DATA_BLOCK "COM_SHUTTLE"	// DB 200
VERSION : 0.1
  STRUCT
   DB_VAR : INT  := 300;	//Temporary placeholder variable
   DB_VAR1 : INT  := 300;	//Temporary placeholder variable
   DB_VAR2 : INT  := 300;	//Temporary placeholder variable
   DB_VAR3 : INT  := 300;	//Temporary placeholder variable
   DB_VAR4 : INT  := 300;	//Temporary placeholder variable
   DB_VAR5 : INT  := 300;	//Temporary placeholder variable
   DB_VAR6 : INT  := 300;	//Temporary placeholder variable
   DB_VAR7 : INT  := 300;	//Temporary placeholder variable
   DB_VAR8 : INT  := 300;	//Temporary placeholder variable
   DB_VAR9 : INT  := 300;	//Temporary placeholder variable
   DB_VAR10 : INT  := 300;	//Temporary placeholder variable
   DB_VAR11 : INT  := 300;	//Temporary placeholder variable
   DB_VAR12 : INT  := 300;	//Temporary placeholder variable
   DB_VAR13 : INT  := 300;	//Temporary placeholder variable
   DB_VAR14 : INT  := 300;	//Temporary placeholder variable
   DB_VAR15 : INT  := 300;	//Temporary placeholder variable
   DB_VAR16 : INT  := 300;	//Temporary placeholder variable
   DB_VAR17 : INT  := 300;	//Temporary placeholder variable
   DB_VAR18 : INT  := 300;	//Temporary placeholder variable
   DB_VAR19 : INT  := 300;	//Temporary placeholder variable
   DB_VAR20 : INT  := 300;	//Temporary placeholder variable
   DB_VAR21 : INT  := 300;	//Temporary placeholder variable
   DB_VAR22 : INT  := 300;	//Temporary placeholder variable
   DB_VAR23 : INT  := 300;	//Temporary placeholder variable
   DB_VAR24 : INT  := 300;	//Temporary placeholder variable
   DB_VAR25 : INT  := 300;	//Temporary placeholder variable
   DB_VAR26 : INT  := 300;	//Temporary placeholder variable
   DB_VAR27 : INT  := 300;	//Temporary placeholder variable
   DB_VAR28 : INT  := 300;	//Temporary placeholder variable
   DB_VAR29 : INT  := 300;	//Temporary placeholder variable
   DB_VAR30 : INT  := 300;	//Temporary placeholder variable
   DB_VAR31 : INT  := 300;	//Temporary placeholder variable
   DB_VAR32 : INT  := 300;	//Temporary placeholder variable
   DB_VAR33 : INT  := 300;	//Temporary placeholder variable
   DB_VAR34 : INT  := 300;	//Temporary placeholder variable
   DB_VAR35 : INT  := 300;	//Temporary placeholder variable
   DB_VAR36 : INT  := 300;	//Temporary placeholder variable
   DB_VAR37 : INT  := 300;	//Temporary placeholder variable
   DB_VAR38 : INT  := 300;	//Temporary placeholder variable
   DB_VAR39 : INT  := 300;	//Temporary placeholder variable
   DB_VAR40 : INT  := 300;	//Temporary placeholder variable
   DB_VAR41 : INT  := 300;	//Temporary placeholder variable
   DB_VAR42 : INT  := 300;	//Temporary placeholder variable
   DB_VAR43 : INT  := 300;	//Temporary placeholder variable
   DB_VAR44 : INT  := 300;	//Temporary placeholder variable
   DB_VAR45 : INT  := 300;	//Temporary placeholder variable
   DB_VAR46 : INT  := 300;	//Temporary placeholder variable
   DB_VAR47 : INT  := 300;	//Temporary placeholder variable
   DB_VAR48 : INT  := 300;	//Temporary placeholder variable
   DB_VAR49 : INT  := 300;	//Temporary placeholder variable
   DB_VAR50 : INT  := 300;	//Temporary placeholder variable
   DB_VAR51 : INT  := 300;	//Temporary placeholder variable
   DB_VAR52 : INT  := 300;	//Temporary placeholder variable
   DB_VAR53 : INT  := 300;	//Temporary placeholder variable
   DB_VAR54 : INT  := 300;	//Temporary placeholder variable
   DB_VAR55 : INT  := 300;	//Temporary placeholder variable
   DB_VAR56 : INT  := 300;	//Temporary placeholder variable
   DB_VAR57 : INT  := 300;	//Temporary placeholder variable
   DB_VAR58 : INT  := 300;	//Temporary placeholder variable
   DB_VAR59 : INT  := 300;	//Temporary placeholder variable
   DB_VAR60 : INT  := 300;	//Temporary placeholder variable
   DB_VAR61 : INT  := 300;	//Temporary placeholder variable
   DB_VAR62 : INT  := 300;	//Temporary placeholder variable
   DB_VAR63 : INT  := 300;	//Temporary placeholder variable
   DB_VAR64 : INT  := 300;	//Temporary placeholder variable
   DB_VAR65 : INT  := 300;	//Temporary placeholder variable
   DB_VAR66 : INT  := 300;	//Temporary placeholder variable
   DB_VAR67 : INT  := 300;	//Temporary placeholder variable
   DB_VAR68 : INT  := 300;	//Temporary placeholder variable
   DB_VAR69 : INT  := 300;	//Temporary placeholder variable
   DB_VAR70 : INT  := 300;	//Temporary placeholder variable
   DB_VAR71 : INT  := 300;	//Temporary placeholder variable
   DB_VAR72 : INT  := 300;	//Temporary placeholder variable
   DB_VAR73 : INT  := 300;	//Temporary placeholder variable
   DB_VAR74 : INT  := 300;	//Temporary placeholder variable
   DB_VAR75 : INT  := 300;	//Temporary placeholder variable
   DB_VAR76 : INT  := 300;	//Temporary placeholder variable
   DB_VAR77 : INT  := 300;	//Temporary placeholder variable
   DB_VAR78 : INT  := 300;	//Temporary placeholder variable
   DB_VAR79 : INT  := 300;	//Temporary placeholder variable
   DB_VAR80 : INT  := 300;	//Temporary placeholder variable
   DB_VAR81 : INT  := 300;	//Temporary placeholder variable
   DB_VAR82 : INT  := 300;	//Temporary placeholder variable
   DB_VAR83 : INT  := 300;	//Temporary placeholder variable
   DB_VAR84 : INT  := 300;	//Temporary placeholder variable
   DB_VAR85 : INT  := 300;	//Temporary placeholder variable
   DB_VAR86 : INT  := 300;	//Temporary placeholder variable
   DB_VAR87 : INT  := 300;	//Temporary placeholder variable
   DB_VAR88 : INT  := 300;	//Temporary placeholder variable
   DB_VAR89 : INT  := 300;	//Temporary placeholder variable
   DB_VAR90 : INT  := 300;	//Temporary placeholder variable
   DB_VAR91 : INT  := 300;	//Temporary placeholder variable
   DB_VAR92 : INT  := 300;	//Temporary placeholder variable
   DB_VAR93 : INT  := 300;	//Temporary placeholder variable
   DB_VAR94 : INT  := 300;	//Temporary placeholder variable
   DB_VAR95 : INT  := 300;	//Temporary placeholder variable
   DB_VAR96 : INT  := 300;	//Temporary placeholder variable
   DB_VAR97 : INT  := 300;	//Temporary placeholder variable
   DB_VAR98 : INT  := 300;	//Temporary placeholder variable
   DB_VAR99 : INT  := 300;	//Temporary placeholder variable
  END_STRUCT ;	
BEGIN
   DB_VAR := 324;
   DB_VAR1 := 3242;
   DB_VAR2 := 2;
   DB_VAR3 := 2;
   DB_VAR4 := 55;
   DB_VAR5 := 1;
   DB_VAR6 := 1;
   DB_VAR7 := 1;
   DB_VAR8 := 1;
   DB_VAR9 := 23423;
   DB_VAR10 := 1;
   DB_VAR11 := 1;
   DB_VAR12 := 1;
   DB_VAR13 := 1;
   DB_VAR14 := 1;
   DB_VAR15 := 2;
   DB_VAR16 := 333;
   DB_VAR17 := 3;
   DB_VAR18 := 300;
   DB_VAR19 := 33;
   DB_VAR20 := 300;
   DB_VAR21 := 8;
   DB_VAR22 := 300;
   DB_VAR23 := 300;
   DB_VAR24 := 300;
   DB_VAR25 := 300;
   DB_VAR26 := 300;
   DB_VAR27 := 4;
   DB_VAR28 := 333;
   DB_VAR29 := 300;
   DB_VAR30 := 300;
   DB_VAR31 := 3;
   DB_VAR32 := 300;
   DB_VAR33 := 300;
   DB_VAR34 := 300;
   DB_VAR35 := 300;
   DB_VAR36 := 4;
   DB_VAR37 := 300;
   DB_VAR38 := 300;
   DB_VAR39 := 300;
   DB_VAR40 := 300;
   DB_VAR41 := 300;
   DB_VAR42 := 300;
   DB_VAR43 := 300;
   DB_VAR44 := 300;
   DB_VAR45 := 300;
   DB_VAR46 := 300;
   DB_VAR47 := 300;
   DB_VAR48 := 300;
   DB_VAR49 := 300;
   DB_VAR50 := 300;
   DB_VAR51 := 300;
   DB_VAR52 := 300;
   DB_VAR53 := 300;
   DB_VAR54 := 300;
   DB_VAR55 := 300;
   DB_VAR56 := 300;
   DB_VAR57 := 300;
   DB_VAR58 := 300;
   DB_VAR59 := 300;
   DB_VAR60 := 300;
   DB_VAR61 := 300;
   DB_VAR62 := 300;
   DB_VAR63 := 300;
   DB_VAR64 := 300;
   DB_VAR65 := 300;
   DB_VAR66 := 300;
   DB_VAR67 := 300;
   DB_VAR68 := 300;
   DB_VAR69 := 300;
   DB_VAR70 := 300;
   DB_VAR71 := 300;
   DB_VAR72 := 300;
   DB_VAR73 := 300;
   DB_VAR74 := 300;
   DB_VAR75 := 300;
   DB_VAR76 := 300;
   DB_VAR77 := 300;
   DB_VAR78 := 300;
   DB_VAR79 := 300;
   DB_VAR80 := 300;
   DB_VAR81 := 300;
   DB_VAR82 := 300;
   DB_VAR83 := 300;
   DB_VAR84 := 300;
   DB_VAR85 := 300;
   DB_VAR86 := 300;
   DB_VAR87 := 300;
   DB_VAR88 := 300;
   DB_VAR89 := 300;
   DB_VAR90 := 300;
   DB_VAR91 := 300;
   DB_VAR92 := 300;
   DB_VAR93 := 300;
   DB_VAR94 := 300;
   DB_VAR95 := 300;
   DB_VAR96 := 300;
   DB_VAR97 := 300;
   DB_VAR98 := 300;
   DB_VAR99 := 300;
END_DATA_BLOCK

DATA_BLOCK "LLOUT"	// DB 201
VERSION : 0.1
  STRUCT
   OUT : STRUCT 	//Dane wejsciowe z Odbierania
    Zadanie_Transmisji : BOOL ;
    Zadanie_Danych : BOOL ;
    Toggle : BOOL ;	//bit- in/out
    Rezerwa_0_3 : BOOL ;
    Rezerwa_0_4 : BOOL ;
    Funcja_Receive : BOOL ;
    Funkcja_Share : BOOL ;
    Rezerwa_0_7 : BOOL ;
    Rezerwa_Bajt_1 : BYTE ;
    Nr_Bloku : INT  := 701;	//Nr bloku gdzie dane (read/send)
    Nr_Rekordu : INT ;	//Nr rekordu wysylanego (read/send)
    Kanal_Nadawania : INT ;	//Kanal Nadawania (send)
    Rezerwa_Bajtow : ARRAY  [1 .. 24 ] OF BYTE ;
   END_STRUCT ;
  END_STRUCT ;	
BEGIN
   OUT.Nr_Bloku := 701;
END_DATA_BLOCK

DATA_BLOCK "LLIN"	// DB 202
VERSION : 0.1
  STRUCT
   IN : STRUCT 	//Dane wejsciowe z Odbierania
    Transmisja_Ustanowiona : BOOL ;
    Blok_Zarezerwowany : BOOL ;
    Toggle : BOOL ;	//bit- in/out
    Przesylanie_Danych : BOOL ;
    Koniec_Nadawania : BOOL ;
    Receive_Wybrane : BOOL ;
    Share_Wybrane : BOOL ;
    Rezerwa_0_7 : BOOL ;
    Rezerwa_Bajt_1 : BYTE ;
    Nr_Rekordu : INT  := 701;
    Licznik_Rekordow : INT ;	//Potwierdzenie Rekordu (Share/receive)
    Kanal_Pobierania : INT ;	//Pobieranie danych (Share)
    Rezerwa_Bajtow : ARRAY  [1 .. 24 ] OF BYTE ;
   END_STRUCT ;
  END_STRUCT ;	
BEGIN
   IN.Nr_Rekordu := 701;
END_DATA_BLOCK

DATA_BLOCK "Stale_Maszynowe"	// DB 300
VERSION : 0.1
  STRUCT
   Pozycja_Skrajna_Dol : DINT  := L#280;
   Pozycja_KB1 : DINT  := L#400;	//Temporary placeholder variable
   Pozycja_KB2 : DINT  := L#15905;
   Pozycja_Gender : DINT  := L#24780;
   Pozycja_odbieranie : DINT  := L#33000;
   Pozycja_Pob_I1 : DINT  := L#34180;
   Pozycja_Skrajna_Gora : DINT  := L#34210;
   Reserwa : DINT ;
   War_W_Kolejce_KB1 : DINT  := L#200;
   War_W_Kolejce_KB2 : DINT  := L#200;
   War_W_Kolejce_I1 : DINT  := L#100;
   War_W_Kolejce_I2 : DINT  := L#100;
   War_W_Kolejce_I3 : DINT  := L#100;
   Pozycja_Pob_I2 : DINT  := L#32944;
   Pozycja_Pob_I3 : DINT  := L#34111;
   Reserwa_21 : DINT ;
   Reserwa_22 : DINT ;
   Reserwa_24 : DINT ;
   res : DINT ;
   res1 : DINT ;
   res2 : DINT ;
   res3 : DINT ;
   res4 : DINT ;
   res5 : DINT ;
   res6 : DINT ;
   res7 : DINT ;
   res8 : DINT ;
   res81 : DINT ;
   res82 : DINT ;
   res83 : DINT ;
   res84 : DINT ;
   res85 : DINT ;
   res86 : DINT ;
   res87 : DINT ;
   res88 : DINT ;
   res89 : DINT ;
   res810 : DINT ;
   res811 : DINT ;
   res812 : DINT ;
   res813 : DINT ;
   res814 : DINT ;
   res815 : DINT ;
   res816 : DINT ;
   res817 : DINT ;
   res818 : DINT ;
   res819 : DINT ;
   res820 : DINT ;
   res821 : DINT ;
   res822 : DINT ;
   res823 : DINT ;
  END_STRUCT ;	
BEGIN
   Pozycja_Skrajna_Dol := L#280;
   Pozycja_KB1 := L#400;
   Pozycja_KB2 := L#15905;
   Pozycja_Gender := L#24780;
   Pozycja_odbieranie := L#33000;
   Pozycja_Pob_I1 := L#34180;
   Pozycja_Skrajna_Gora := L#34210;
   War_W_Kolejce_KB1 := L#200;
   War_W_Kolejce_KB2 := L#200;
   War_W_Kolejce_I1 := L#100;
   War_W_Kolejce_I2 := L#100;
   War_W_Kolejce_I3 := L#100;
   Pozycja_Pob_I2 := L#32944;
   Pozycja_Pob_I3 := L#34111;
END_DATA_BLOCK

DATA_BLOCK "Key_DB"	// DB 409
VERSION : 0.1
  STRUCT
   Wpis : STRUCT
    _0_dbb0_Kod_Kier : BYTE ;
    _0_dbb1_Kod_Maszyna : BYTE ;
    _0_dbw2_War_Wagowa : INT ;
    _1_dbb4_Kod_Kier : BYTE ;
    _1_dbb5_Kod_Maszyna : BYTE ;
    _1_dbw6_War_Wagowa : INT ;
    _2_dbb8_Kod_Kier : BYTE ;
    _2_dbb9_Kod_Maszyna : BYTE ;
    _2_dbw10_War_Wagowa : INT ;
    _3_dbb12_Kod_Kier : BYTE ;
    _3_dbb13_Kod_Maszyna : BYTE ;
    _3_dbw14_War_Wagowa : INT ;
    _4_dbb16_Kod_Kier : BYTE ;
    _4_dbb17_Kod_Maszyna : BYTE ;
    _4_dbw18_War_Wagowa : INT ;
    _5_dbb20_Kod_Kier : BYTE ;
    _5_dbb21_Kod_Masz : BYTE ;
    _5_dbw22_War_Wagowa : INT ;
    _6_dbb24_Kod_Kier : BYTE ;
    _6_dbb25_Kod_Masz : BYTE ;
    _6_dbw26_War_Wagowa : INT ;
    Kod_Spr_KB1 : BYTE ;
    Kod_Spr_KB2 : BYTE ;
    Kod_Spr_I1 : BYTE ;
    Kod_Spr_I2 : BYTE ;
    Kod_Spr_I3 : BYTE ;
    Kod_Spr_Rezerwa : BYTE ;
   END_STRUCT ;
  END_STRUCT ;	
BEGIN
   Wpis._3_dbw14_War_Wagowa := 200;
END_DATA_BLOCK

ORGANIZATION_BLOCK OB 1
TITLE = "Main Program Sweep (Cycle)"
VERSION : 0.1
VAR_TEMP
  OB1_EV_CLASS : BYTE ;	//Bits 0-3 = 1 (Coming event), Bits 4-7 = 1 (Event class 1)
  OB1_SCAN_1 : BYTE ;	//1 (Cold restart scan 1 of OB 1), 3 (Scan 2-n of OB 1)
  OB1_PRIORITY : BYTE ;	//Priority of OB Execution
  OB1_OB_NUMBR : BYTE ;	//1 (Organization block 1, OB1)
  OB1_RESERVED_1 : BYTE ;	//Reserved for system
  OB1_RESERVED_2 : BYTE ;	//Reserved for system
  OB1_PREV_CYCLE : INT ;	//Cycle time of previous OB1 scan (milliseconds)
  OB1_MIN_CYCLE : INT ;	//Minimum cycle time of OB1 (milliseconds)
  OB1_MAX_CYCLE : INT ;	//Maximum cycle time of OB1 (milliseconds)
  OB1_DATE_TIME : DATE_AND_TIME ;	//Date and time OB1 started
END_VAR
BEGIN
NETWORK
TITLE =
      CALL  "Wozek_Jezdny_Kolejka";
END_ORGANIZATION_BLOCK

ORGANIZATION_BLOCK "PROG_ERR"	// OB 121
TITLE = "Programming Error"
VERSION : 0.1
VAR_TEMP
  OB121_EV_CLASS : BYTE ;	//16#25, Event class 2, Entering event state, Internal fault event
  OB121_SW_FLT : BYTE ;	//16#XX Software programming fault
  OB121_PRIORITY : BYTE ;	//Priority of OB Execution
  OB121_OB_NUMBR : BYTE ;	//121 (Organization block 121, OB121)
  OB121_BLK_TYPE : BYTE ;	//16#88/8A/8B/8C/8E Type of block fault occured in
  OB121_RESERVED_1 : BYTE ;	//Reserved for system
  OB121_FLT_REG : WORD ;	//16#XX Specific register that caused fault
  OB121_BLK_NUM : WORD ;	//Number of block that programming fault occured in
  OB121_PRG_ADDR : WORD ;	//Address in block where programming fault occured
  OB121_DATE_TIME : DATE_AND_TIME ;	//Date and time OB121 started
END_VAR
BEGIN
// (block stored without names or comments; labels and parameter names are numbered)
END_ORGANIZATION_BLOCK

SYMBOL_TABLE
"Licznik_1"	C 1	COUNTER
"Blok_Bledow"	DB 119	DB 119
"COM_ODB"	DB 200	DB 200	// Blok komunikacji odbieranie shuttle
"LIN"	DB 201	DB 201
"LOUT"	DB 202	DB 202	// Blok wymiany danych dlugi
"Blok_Parametrow"	DB 701	DB 701
"Blok_Stref_Kier_KB1"	DB 720	DB 720	// Blok zawierajacy pozycje i strefe przyporzadkowana
"Blok_Stref_Kier_Rot"	DB 721	DB 721
"Funkcja_Bezpieczenstwa"	FC 3	FC 3
"Fal_Lenze_V_3"	FC 10	FC 10
"Zasprzeglenie_Bandy"	FC 30	FC 30
"Funkcja_Wymiany_Danych"	FC 40	FC 40
"Odbieranie_Danych"	FC 41	FC 41
"Wysylanie_Danych"	FC 42	FC 42
"Aufruf Achse 1"	FC 100	FC 100
"Jazda_Shuttle"	FC 101	FC 101
"Przelaczanie_Stref_K_Rot"	FC 102	FC 102	// Przelaczanie Stref kierunek KB1-Rotacja
"Przelaczanie_Stref_K_KB1"	FC 103	FC 103
"Blok_Bedow"	FC 119	FC 119
"Fal_Sew"	FC 140	FC 140	// Falownik Sew wersja niemiecka funkcji
"Predkosc_Fal"	FC 141	FC 141	// Funkcja  doboru predkosci
"Funkcja_Zegara"	FC 150	FC 150	// Funkcja zegara
"COM_Odbieranie"	FC 200	FC 200
"COM_Pakiety"	FC 201	FC 201	// Odbieranie i wysylanie pakietow danych
"Receive_Data"	FC 701	FC 701
"Share_Data"	FC 703	FC 703	// Funkcja udostepniajaca dane
"Bezp_OK"	I 4.0	BOOL	// Bezpieczniki ok Shuttle [ I4.0 s.10 ]
"Przekaznik_Bezp_Ok"	I 4.1	BOOL	// Przekaznik Bezpieczenstwa OK [I4.1 s.10]
"Listwa_Bezp_OK"	I 4.2	BOOL	// Listwa Bezpieczenstwa OK [I4.2 s. 10]
"PB_Auto_Reczny"	I 4.3	BOOL	// Auto reczny kaseta [I4.4 s.10]
"PB_Rewizja"	I 4.4	BOOL	// Rewizja kaseta [I4.4 s. 10]
"PB_Reset_Kaseta"	I 4.5	BOOL	// Reset kaseta [I4.5 s. 10]
"PB_Jazda_Przod"	I 4.6	BOOL	// Jazda Tyl kaseta [I4.6 s. 10]
"PB_Jazda_Tyl"	I 4.7	BOOL	// Jazda Tyl kaseta [I4.7 s. 10]
"Przekaznik_Bezp_Rewizja"	I 5.0	BOOL	// Przekaznik Rewizja OK [I5.0 s. 12]
"Rezerwa_I5.1"	I 5.1	BOOL
"Foto_Banda_Przod"	I 5.2	BOOL	// Fotokomorka Banda Przod [I5.2 s. 11]
"Foto_Banda_Tyl"	I 5.3	BOOL	// Fotokomorka Banda Tyl [I5.3 s. 11]
"Czujnik_Poz_Ham"	I 5.4	BOOL	// Czujnik pozycji hamowania [I5.3 s. 11]
"Czujnik_Shuttle_Na_Poz"	I 5.5	BOOL	// Czujnik shuttle na pozycji [I5.5  s. 11]
"Ham_Reczny_Zalaczony"	I 5.6	BOOL	// Przelacznik_Hamulca_Zalaczony [I5.6 s.11]
"Reset_Przek_Bezp_Wozek"	I 5.7	BOOL	// Reset przekaznik bezp wozek [I5.7 s.11]
"Skaner_P_Strefa_Ostrz"	I 6.0	BOOL	// Skaner przedni strefa ostrzegawcza [I6.0 s 12]
"Skaner_P_Reset_Wym"	I 6.1	BOOL	// Skaner przedni reset wymagany [I6.1 s. 12]
"Skaner_P_Error"	I 6.2	BOOL	// Skaner przedni error  [I6.2 s. 12]
"Skaner_P_Strefa_OK"	I 6.3	BOOL	// Skaner przeni strefa OK [I6.3 s. 12]
"Rezerwa_6.4"	I 6.4	BOOL
"Rezerwa_6.5"	I 6.5	BOOL
"Rezerwa_6.6"	I 6.6	BOOL
"Rezerwa_6.7"	I 6.7	BOOL
"Skaner_T_Strefa_Ostrz"	I 7.0	BOOL	// Skaner tylni strefa ostrzegawcza [I7.0 s 13]
"Skaner_T_Reset_Wym"	I 7.1	BOOL	// Skaner tylni reset wymagany [I7.1 s. 13]
"Skaner_T_Error"	I 7.2	BOOL	// Skaner tylni error  [I7.2 s. 13]
"Skaner_T_Strefa_OK"	I 7.3	BOOL	// Skaner tylni strefa OK [I7.3 s. 13]
"Rezerwa_7.4"	I 7.4	BOOL
"Rezerwa_7.5"	I 7.5	BOOL
"Rezerwa_7.6"	I 7.6	BOOL
"Rezerwa_7.7"	I 7.7	BOOL
"Zez_Demag"	I 8.0	BOOL	// Petla Do Demago OK
"Zew_Not_Aus_OK"	I 8.1	BOOL	// Zewnetrzne Not-Aus OK [I8.1 s. 14]
"Sygnaly_Wejsciowe"	ID 38	DWORD	// Sygnaly wejsciowe shuttle
"Pozycja zadana"	ID 42	DINT	// -->Pozycja Zadana Shuttle
"Zawsze_True"	M 0.0	BOOL
"Zawsze_False"	M 0.1	BOOL
"Reset_Wozka"	M 0.2	BOOL
"Marka_Bladzaca"	M 0.3	BOOL
"Reset_Bledow"	M 0.4	BOOL
"Auto_Reczny"	M 1.0	BOOL	// Shuttle Auto-Reczny
"Marka_Bezpieczenstwa_0"	M 2.0	BOOL
"Marka_Bezpieczenstwa_1"	M 2.1	BOOL
"Miganie_200ms"	M 10.0	BOOL
"Miganie_500ms"	M 10.1	BOOL
"Miganie_100ms"	M 10.2	BOOL
"Reset_Bledu_Silnika"	M 11.0	BOOL
"Sygnal_Przedstartu"	M 11.1	BOOL
"M_Zezwolenie_Bandy"	M 20.0	BOOL	// Zezwolenie jazda band
"Silnik_Lewo"	M 20.1	BOOL
"Silnik_Prawo"	M 20.2	BOOL
"Start_Silnika"	M 20.3	BOOL
"Silnik_Lewo_Prawo"	M 20.4	BOOL
"Odblokuj_Lenze"	M 20.5	BOOL
"Falownik_Gotowy"	M 20.6	BOOL
"Falownik_Blad"	M 20.7	BOOL
"Hamulec_Lenze"	M 21.0	BOOL
"Blokada_Jazdy_W_Prawo"	M 21.1	BOOL
"Blokada_Jazdy_W_Lewo"	M 21.2	BOOL
"Blokada_Lewo"	M 21.3	BOOL
"Blokada_Prawo"	M 21.4	BOOL
"Pokrycie_Foto_Ok"	M 21.5	BOOL
"Jedz_Na_nowa_Pozycje"	M 40.0	BOOL
"Brak_Kom_Odbieranie"	M 40.2	BOOL
"Shutte_Stoi"	M 40.3	BOOL	// Wozek nie jedzie
"Wozek_Zasprzeglony"	M 40.4	BOOL
"Wozek_Rozprzeglony"	M 40.5	BOOL
"Silnik_Band_Stoi"	M 40.6	BOOL
"Shuttle_Wypozycjonowany"	M 42.0	BOOL
"Wypozycj_1_Stopien"	M 42.1	BOOL
"Marka_Startu"	M 99.0	BOOL
"Zez_Jazda_Wozek"	M 100.0	BOOL
"Reset_Blad_Wozek"	M 100.1	BOOL
"Jog_Plus_Wozek"	M 100.2	BOOL
"Jog_Minus_Wozek"	M 100.3	BOOL
"Tryb_Referencji"	M 100.4	BOOL
"Tryb_Pozycjonowania"	M 100.5	BOOL
"Komunikacja_Fal_Ok"	M 101.0	BOOL
"Blad_Os_Wozek"	M 101.1	BOOL
"Ostrz_Os_Wozek"	M 101.2	BOOL
"Falownik_Wozek_Gotowy"	M 101.3	BOOL
"Wozek_W_Referencji"	M 101.4	BOOL
"OS_Wozek_Zablokowana"	M 101.6	BOOL
"Pozycja_Jazdy_Osiagnieta"	M 101.7	BOOL
"Jazda_Kier_Rot"	M 122.0	BOOL
"Jazda_Kier_KB1"	M 122.1	BOOL
"Sygnal_Przedni"	M 122.2	BOOL
"Sygnal_Tylni"	M 122.3	BOOL
"Help_M122.7"	M 122.7	BOOL
"MI_Zadanie_Transmisji"	M 428.0	BOOL
"MI_Zadanie_Danych"	M 428.1	BOOL
"MI_Toggle"	M 428.2	BOOL
"MI_0_3"	M 428.3	BOOL
"MI_0_4"	M 428.4	BOOL
"MI_Funcja_Receive"	M 428.5	BOOL
"MI_Funkcja_Share"	M 428.6	BOOL
"MI_0_7"	M 428.7	BOOL
"Toggle_Para"	M 501.1	BOOL
"MO_Trans_Ustawiona"	M 528.0	BOOL
"MO_Blok_Zarez"	M 528.1	BOOL
"M_Przesylanie_Danych"	M 528.3	BOOL
"MO_Koniec_Nadawania"	M 528.4	BOOL
"MO_Receive_Wybrane"	M 528.5	BOOL
"MO_Share_Wybrane"	M 528.6	BOOL
"MO_0_7"	M 528.7	BOOL
"MIB_1_0"	MB 429	BYTE
"MOB_529"	MB 529	BYTE
"Predkosc_Tasmy"	MD 22	REAL
"Predkosc_Transportera"	MD 26	REAL
"Pozycja_Zadana"	MD 436	DINT
"Pozycja_Aktualna"	MD 536	DINT
"Falownik_STW"	MW 22	WORD
"Waga_Licznika"	MW 60	INT
"Predkosc_Zadana"	MW 106	INT
"Rampa_Startowa"	MW 108	INT
"Rampa_Zatrzymania"	MW 110	INT
"Nr_Bledu_Wozek"	MW 112	INT
"Predkosc_Aktualna"	MW 118	INT
"Prad_Aktualny"	MW 120	INT
"Predk_Wozka_K_KB1_Rot"	MW 124	INT
"Predk_Wozka_Kier_KB1"	MW 128	INT
"Predkosc_Ostrzegawcza"	MW 140	INT
"Predkosc_Pod_Obciazeniem"	MW 144	INT
"Zaleznosc_Od_Skanerow"	MW 146	INT
"Predkosc_Cargo"	MW 148	INT
"Predkosc_Maks_Wozek"	MW 200	INT
"MIW_Nr_Bloku"	MW 430	INT
"MIW_Kanal_Odbioru"	MW 432	WORD
"MIW_Licznik_Rekordow"	MW 434	INT
"Help_MW_490"	MW 490	WORD
"Help_mw_492"	MW 492	WORD
"MOW_Nr_Rekordu"	MW 530	INT
"MOW_Kanal_Pobierania"	MW 532	WORD
"Predkosc_Aktualna_Wozka"	MW 540	INT
"Licznik_Rekordu"	MW 600	INT
"Program_Glowny"	OB 1	OB 1
"I/O_FLT1"	OB 82	OB 82	// I/O Point Fault 1
"RACK_FLT"	OB 86	OB 86	// Loss of Rack Fault
"PROG_ERR"	OB 121	OB 121	// Programming Error
"MOD_ERR"	OB 122	OB 122	// Module Access Error
"Syrena_Ton_1"	Q 12.0	BOOL	// Syrena ton 1 [q12.0 s. 18]
"Syrena_Ton_2"	Q 12.1	BOOL	// Syrena ton 2 [q12.1 s. 18]
"Zasilanie_Foto"	Q 12.2	BOOL	// Zasilanie Fotokomorek[q12.2 s. 18]
"Reset_P_Bezpieczenstwa"	Q 12.3	BOOL	// Reset przekaznika bezpieczenstwa [q12.3 s. 18]
"Zez_Transport_Shuttle"	Q 12.4	BOOL	// Zezwolenie na jazde SHuttle [q12.4 s. 18]
"Zez_Transport_Przenosnik"	Q 12.5	BOOL	// Zezwolenie na transport przenosnik [q12.5 s. 18]
"Zez_Rewizja_1"	Q 12.6	BOOL	// Zezwolenie rewizja 1 [q12.6 s. 18]
"Zez_Rewizja_2"	Q 12.7	BOOL	// Zezwolenie rewizja 2 [q12.7 s. 18]
"Lamp_Kier_Przod"	Q 13.0	BOOL	// Kierunkowskazy przednie [q13.0 s. 19]
"Lamp_Kier_Tyl"	Q 13.1	BOOL	// Kierunkowskazy tylne [q13.1 s. 19]
"Lamp_Wieza_Zielony"	Q 13.2	BOOL	// Lampa wieza sygnalizacyjna czerwony [q13.5 s. 19]
"Lamp_Wieza_Pom"	Q 13.3	BOOL	// Lampa wieza sygnalizacyjna pomaranczowy [q13.4 s. 19]
"Lamp_Wieza_Czerw"	Q 13.4	BOOL	// Lampa wieza sygnalizacyjna zielony [q13.3 s. 19]
"Lamp_Wieza_Bialy"	Q 13.5	BOOL	// Lampa wieza sygnalizacyjna niebieski  zasprzeglenie [q13.6 s. 19]
"Lamp_Wieza_Syrena"	Q 13.6	BOOL	// Syrena wieza sygnalizacyjna [q13.2 s. 19]
"Sygn_Wieza"	Q 13.7	BOOL	// Lampa przejazdu pomaranczowa [q13.7 s. 19]
"Skaner_P_Reset"	Q 14.0	BOOL	// Skaner przedni reset [q14.0 s. 20]
"Skaner_P_Strefa_1"	Q 14.1	BOOL	// Skaner przedni strefa 1[ q14.1 s. 20]
"Skaner_P_Strefa_2"	Q 14.2	BOOL	// Skaner przedni strefa 2[ q14.2 s. 20]
"Skaner_P_Strefa_3"	Q 14.3	BOOL	// Skaner przedni strefa 3[ q14.3 s. 20]
"Skaner_P_Strefa_4"	Q 14.4	BOOL	// Skaner przedni strefa 4[ q14.4 s. 20]
"Zar_PB_Reset"	Q 14.5	BOOL	// ¯arowka Reset [q14.6 s.20]
"Reserwa_Q14.6"	Q 14.6	BOOL
"Hamulec_Rolki"	Q 14.7	BOOL	// Hamulec Lenze Rolki  [ q14.7 s. 20]
"Skaner_T_Reset"	Q 15.0	BOOL	// Skaner tylni reset [q15.0 s. 21]
"Skaner_T_Strefa_1"	Q 15.1	BOOL	// Skaner tylni strefa 1[ q15.1 s. 21]
"Skaner_T_Strefa_2"	Q 15.2	BOOL	// Skaner tylni strefa 2[ q15.2 s. 21]
"Skaner_T_Strefa_3"	Q 15.3	BOOL	// Skaner tylni strefa 3[ q15.3 s. 21]
"Skaner_T_Strefa_4"	Q 15.4	BOOL	// Skaner tylni strefa 4[ q15.4 s. 21]
"Rezerwa_Q11.5"	Q 15.5	BOOL
"Rezerwa_Q11.6"	Q 15.6	BOOL
"Rezerwa_Q11.7"	Q 15.7	BOOL
"DWORD_0_Odbieranie"	QD 30	DWORD
"DWORD_4_Odbieranie"	QD 34	DWORD
"BLKMOV"	SFC 20	SFC 20	// Copy Variables
"Timer_T5"	T 5	TIMER
"Timer_T8"	T 8	TIMER
"Czas_Opoz_Startu_T10"	T 10	TIMER
"Czas_T11"	T 11	TIMER
"Czas_T12"	T 12	TIMER
"Timer_16"	T 16	TIMER
"Timmer_T17"	T 17	TIMER
"Timmer_18"	T 18	TIMER
"T20"	T 20	TIMER
"Miganie_T31"	T 31	TIMER
"Miganie_T32"	T 32	TIMER
"Miganie_T33"	T 33	TIMER
"T40"	T 40	TIMER
"T41"	T 41	TIMER
"T42"	T 42	TIMER
"erweiterte Busposi."	VAT 1	
"VAT_Strefy"	VAT 2	
END_SYMBOL_TABLE

FUNCTION "Funkcja_Bezpieczenstwa" : VOID	// FC 3
VERSION : 0.1
BEGIN
NETWORK
TITLE =
//Ten Network celowo jest wolny
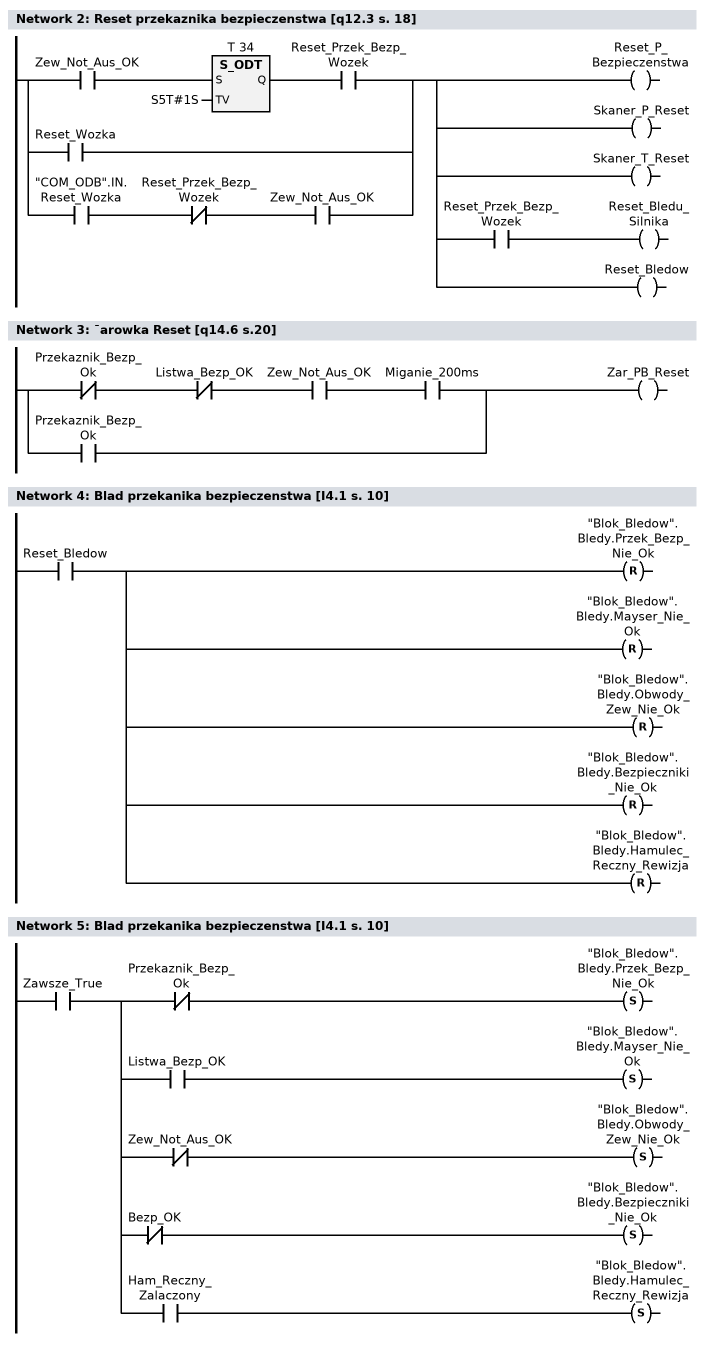
NETWORK
TITLE = Reset przekaznika bezpieczenstwa [q12.3 s. 18]
//Reset przekaznika bezpieczenstwa
      A(;
      A     "Zew_Not_Aus_OK";
      L     S5T#1S;
      SD    T 34;
      NOP   0;
      NOP   0;
      NOP   0;
      A     T 34;
      );
      A     "Reset_Przek_Bezp_Wozek";
      O     "Reset_Wozka";
      O;
      A     "COM_ODB".IN.Reset_Wozka;
      AN    "Reset_Przek_Bezp_Wozek";
      A     "Zew_Not_Aus_OK";
      =     L 0.0;
      A     L 0.0;
      BLD   102;
      =     "Reset_P_Bezpieczenstwa";
      A     L 0.0;
      BLD   102;
      =     "Skaner_P_Reset";
      A     L 0.0;
      BLD   102;
      =     "Skaner_T_Reset";
      A     L 0.0;
      A     "Reset_Przek_Bezp_Wozek";
      =     "Reset_Bledu_Silnika";
      A     L 0.0;
      BLD   102;
      =     "Reset_Bledow";
NETWORK
TITLE = ¯arowka Reset [q14.6 s.20]
//Sprawdzenie czy petla obwodow jest do potwierdzenia
      AN    "Przekaznik_Bezp_Ok";
      AN    "Listwa_Bezp_OK";
      A     "Zew_Not_Aus_OK";
      A     "Miganie_200ms";
      O     "Przekaznik_Bezp_Ok";
      =     "Zar_PB_Reset";
NETWORK
TITLE = Blad przekanika bezpieczenstwa [I4.1 s. 10]
//Reset bledow
      A     "Reset_Bledow";
      R     "Blok_Bledow".Bledy.Przek_Bezp_Nie_Ok;
      R     "Blok_Bledow".Bledy.Mayser_Nie_Ok;
      R     "Blok_Bledow".Bledy.Obwody_Zew_Nie_Ok;
      R     "Blok_Bledow".Bledy.Bezpieczniki_Nie_Ok;
      R     "Blok_Bledow".Bledy.Hamulec_Reczny_Rewizja;
NETWORK
TITLE = Blad przekanika bezpieczenstwa [I4.1 s. 10]
//Przekaznik bezpieczenstwa nie ok
      A     "Zawsze_True";
      =     L 0.0;
      A     L 0.0;
      AN    "Przekaznik_Bezp_Ok";
      S     "Blok_Bledow".Bledy.Przek_Bezp_Nie_Ok;
      A     L 0.0;
      A     "Listwa_Bezp_OK";
      S     "Blok_Bledow".Bledy.Mayser_Nie_Ok;
      A     L 0.0;
      AN    "Zew_Not_Aus_OK";
      S     "Blok_Bledow".Bledy.Obwody_Zew_Nie_Ok;
      A     L 0.0;
      AN    "Bezp_OK";
      S     "Blok_Bledow".Bledy.Bezpieczniki_Nie_Ok;
      A     L 0.0;
      A     "Ham_Reczny_Zalaczony";
      S     "Blok_Bledow".Bledy.Hamulec_Reczny_Rewizja;
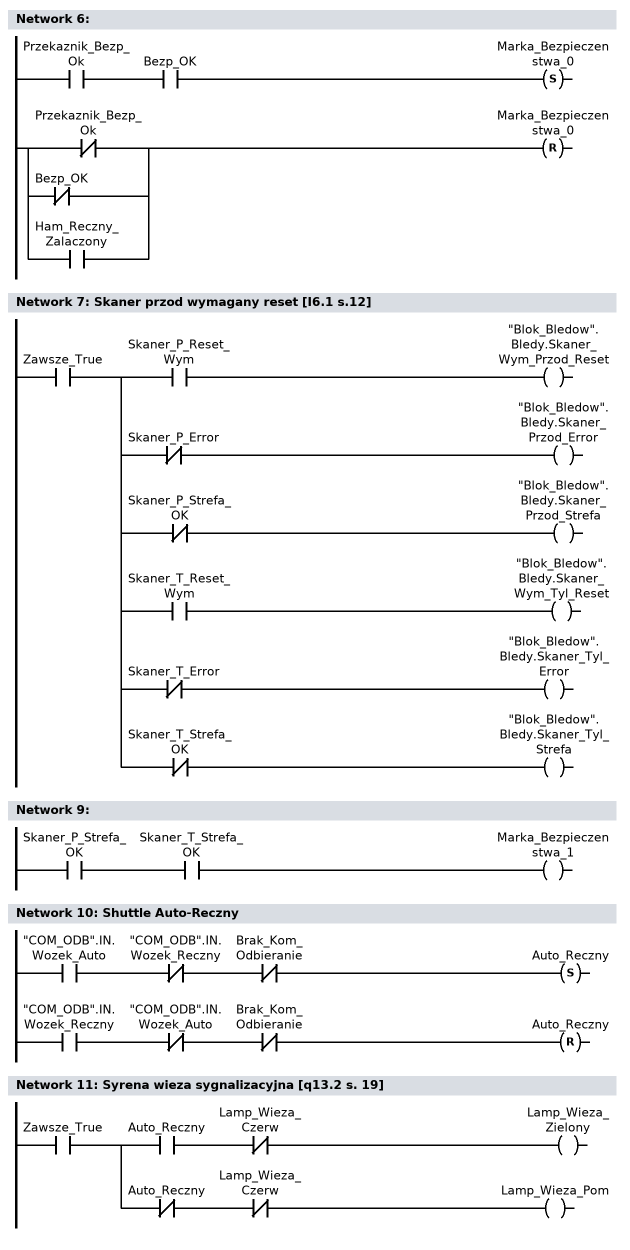
NETWORK
TITLE =
//Sprawdzenie przekaznika bezpieczenswa
//
      A     "Przekaznik_Bezp_Ok";
      A     "Bezp_OK";
      S     "Marka_Bezpieczenstwa_0";
      A(;
      ON    "Przekaznik_Bezp_Ok";
      ON    "Bezp_OK";
      O     "Ham_Reczny_Zalaczony";
      );
      R     "Marka_Bezpieczenstwa_0";
      NOP   0;
NETWORK
TITLE = Skaner przod wymagany reset [I6.1 s.12]
//Bledy skanerow. Kwituja sie same.
      A     "Zawsze_True";
      =     L 0.0;
      A     L 0.0;
      A     "Skaner_P_Reset_Wym";
      =     "Blok_Bledow".Bledy.Skaner_Wym_Przod_Reset;
      A     L 0.0;
      AN    "Skaner_P_Error";
      =     "Blok_Bledow".Bledy.Skaner_Przod_Error;
      A     L 0.0;
      AN    "Skaner_P_Strefa_OK";
      =     "Blok_Bledow".Bledy.Skaner_Przod_Strefa;
      A     L 0.0;
      A     "Skaner_T_Reset_Wym";
      =     "Blok_Bledow".Bledy.Skaner_Wym_Tyl_Reset;
      A     L 0.0;
      AN    "Skaner_T_Error";
      =     "Blok_Bledow".Bledy.Skaner_Tyl_Error;
      A     L 0.0;
      AN    "Skaner_T_Strefa_OK";
      =     "Blok_Bledow".Bledy.Skaner_Tyl_Strefa;
NETWORK
TITLE =
NETWORK
TITLE =
//Petla bezpieczenstwa 1
      A     "Skaner_P_Strefa_OK";
      A     "Skaner_T_Strefa_OK";
      =     "Marka_Bezpieczenstwa_1";
NETWORK
TITLE = Shuttle Auto-Reczny
//Wozek Auto_Reczny
      A     "COM_ODB".IN.Wozek_Auto;
      AN    "COM_ODB".IN.Wozek_Reczny;
      AN    "Brak_Kom_Odbieranie";
      S     "Auto_Reczny";
      A     "COM_ODB".IN.Wozek_Reczny;
      AN    "COM_ODB".IN.Wozek_Auto;
      AN    "Brak_Kom_Odbieranie";
      R     "Auto_Reczny";
      NOP   0;
NETWORK
TITLE = Syrena wieza sygnalizacyjna [q13.2 s. 19]
//Wozek automatyka reczny
      A     "Zawsze_True";
      =     L 0.0;
      A     L 0.0;
      A     "Auto_Reczny";
      AN    "Lamp_Wieza_Czerw";
      =     "Lamp_Wieza_Zielony";
      A     L 0.0;
      AN    "Auto_Reczny";
      AN    "Lamp_Wieza_Czerw";
      =     "Lamp_Wieza_Pom";
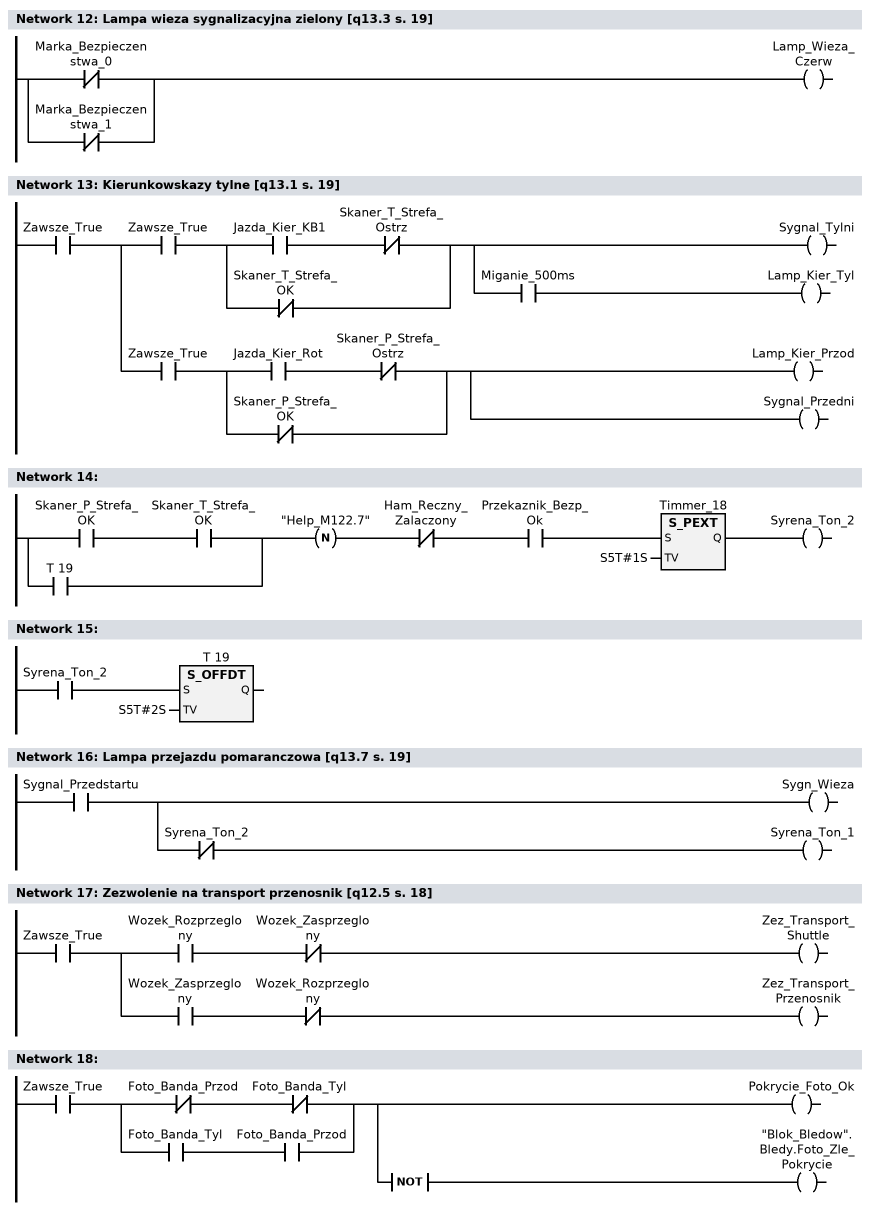
NETWORK
TITLE = Lampa wieza sygnalizacyjna zielony [q13.3 s. 19]
//Lampka wieza czerwona
      ON    "Marka_Bezpieczenstwa_0";
      ON    "Marka_Bezpieczenstwa_1";
      =     "Lamp_Wieza_Czerw";
NETWORK
TITLE = Kierunkowskazy tylne [q13.1 s. 19]
//kierunkowskazy przednie
      A     "Zawsze_True";
      =     L 0.0;
      A     L 0.0;
      A     "Zawsze_True";
      A(;
      A     "Jazda_Kier_KB1";
      AN    "Skaner_T_Strefa_Ostrz";
      ON    "Skaner_T_Strefa_OK";
      );
      =     L 0.1;
      A     L 0.1;
      BLD   102;
      =     "Sygnal_Tylni";
      A     L 0.1;
      A     "Miganie_500ms";
      =     "Lamp_Kier_Tyl";
      A     L 0.0;
      A     "Zawsze_True";
      A(;
      A     "Jazda_Kier_Rot";
      AN    "Skaner_P_Strefa_Ostrz";
      ON    "Skaner_P_Strefa_OK";
      );
      =     "Lamp_Kier_Przod";
      =     "Sygnal_Przedni";
NETWORK
TITLE =
      A(;
      A     "Skaner_P_Strefa_OK";
      A     "Skaner_T_Strefa_OK";
      O     T 19;
      );
      FN    "Help_M122.7";
      AN    "Ham_Reczny_Zalaczony";
      A     "Przekaznik_Bezp_Ok";
      L     S5T#1S;
      SE    "Timmer_18";
      NOP   0;
      NOP   0;
      NOP   0;
      A     "Timmer_18";
      =     "Syrena_Ton_2";
NETWORK
TITLE =
      A     "Syrena_Ton_2";
      L     S5T#2S;
      SF    T 19;
      NOP   0;
      NOP   0;
      NOP   0;
      NOP   0;
NETWORK
TITLE = Lampa przejazdu pomaranczowa [q13.7 s. 19]
//Swiecenie wozka podczas jazdy
      A     "Sygnal_Przedstartu";
      =     L 0.0;
      A     L 0.0;
      BLD   102;
      =     "Sygn_Wieza";
      A     L 0.0;
      AN    "Syrena_Ton_2";
      =     "Syrena_Ton_1";
NETWORK
TITLE = Zezwolenie na transport przenosnik [q12.5 s. 18]
//Zezwolenia do silników
//
      A     "Zawsze_True";
      =     L 0.0;
      A     L 0.0;
      A     "Wozek_Rozprzeglony";
      AN    "Wozek_Zasprzeglony";
      =     "Zez_Transport_Shuttle";
      A     L 0.0;
      A     "Wozek_Zasprzeglony";
      AN    "Wozek_Rozprzeglony";
      =     "Zez_Transport_Przenosnik";
NETWORK
TITLE =
//Sprawdzenie pokrycie fotokomorek
      A     "Zawsze_True";
      A(;
      AN    "Foto_Banda_Przod";
      AN    "Foto_Banda_Tyl";
      O;
      A     "Foto_Banda_Tyl";
      A     "Foto_Banda_Przod";
      );
      =     L 0.0;
      A     L 0.0;
      BLD   102;
      =     "Pokrycie_Foto_Ok";
      A     L 0.0;
      NOT;
      =     "Blok_Bledow".Bledy.Foto_Zle_Pokrycie;
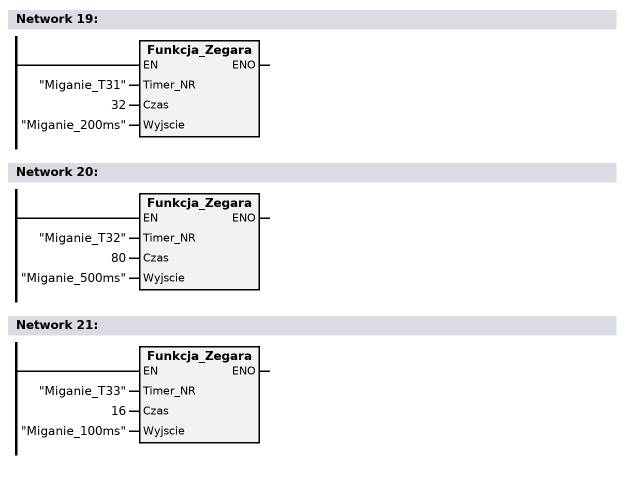
NETWORK
TITLE =
//Timmer generujacy takt 200ms
//
      CALL  "Funkcja_Zegara" (
           Timer_NR                 := "Miganie_T31",
           Czas                     := 32,
           Wyjscie                  := "Miganie_200ms");
      NOP   0;
NETWORK
TITLE =
//Timmer generujacy takt 500ms
      CALL  "Funkcja_Zegara" (
           Timer_NR                 := "Miganie_T32",
           Czas                     := 80,
           Wyjscie                  := "Miganie_500ms");
      NOP   0;
NETWORK
TITLE =
//Timmer generujacy takt 100ms
      CALL  "Funkcja_Zegara" (
           Timer_NR                 := "Miganie_T33",
           Czas                     := 16,
           Wyjscie                  := "Miganie_100ms");
      NOP   0;
END_FUNCTION

FUNCTION "Fal_Lenze_V_3" : VOID	// FC 10
//Funkcja kontrolujaca Falownik Lenze.Zakladane jest ze obszar wejsc falownika 
//pokrywa sie z obszarem wyjsc(PIWX,PQWY,X=Y patrz Hardware).
//
//***CTW***
//POW1-S³owo  kontrolne 1 (CTW)
//POW2-Predkosc zadana (NSET1-N1):+-480HZ=+-24000
//**STW***
//PIW1-S³owo statusu 1 (STW)
//PIW2-Czestotliwosc wyjsciowa+poslizg
//
//
//-Wyroznia sie nastepujace s³owa sterujace:
//CTW:0000 0000 0111 1110 (007E)-falownik gotowy do startu/Funkcja Stop
//CTW:0000 0000 0111 1111 (007F)-falownik zostaje uruchominony
//CTW:xxxx xxxx xxxx x01x (x-wszystko jedno)-falownik zatrzymany Szybki Stop
//-Wyroznia sie nastepujace s³owa statusu:
//STW:xxxx xxxx x01x 0001-Falownik gotowy do startu
//STW:xxxx xxxx x01x 0111-Falownik pracuje
//STW:xxxx xxxx x0xx 1000-Blad Falownika 
//
//
//
AUTHOR : Kng
NAME : DRIVE
VERSION : 0.1
VAR_INPUT
  ADD_Falownika : INT ;
  ESTOP : BOOL ;	//Szybki Stop Falownika
  Start_Lewo : BOOL ;	//Start Falownika CW
  Start_Prawo : BOOL ;	//Start Falownika CCW
  Predkosc_Zadana : REAL ;	//Predkosc silnika w Hz
  Timmer_Pom : INT ;	//Timmer pomocniczy
  Timmer_Pom_2 : INT ;
END_VAR
VAR_OUTPUT
  Falownik_Gotowy : BOOL ;
  Blad_Falownika : BOOL ;	//Falownik zwraca blad
  Odblokuj_Falownik : BOOL ;	//Przekaznik_Odblokowujacy
  Hamulec : BOOL ;	//Odblokowanie hamulca
  Slowo_Statusu : WORD ;	//Slowo Satusu falownika
  Predkosc_zwracana : REAL ;	//Predkosc zwracana przez Falownik
END_VAR
VAR_TEMP
  Adres_1 : DWORD ;
  Adres_2 : DWORD ;
  STW : WORD ;
  CTW : BOOL ;
  H_Temp : INT ;
  H_Temp_2 : INT ;
  Help_Bool_1 : BOOL ;
  Adres_3 : DWORD ;
  Timmer_Name : WORD ;
END_VAR
BEGIN
NETWORK
TITLE =
//Wskaznik do falownika
//********************************Wyliczenie Adresow
      L     #ADD_Falownika;
      SLD   3;
      T     #Adres_1;	//adres falownika control word
      L     #ADD_Falownika;
      L     2;
      +I;
      SLD   3;
      T     #Adres_2;	//adres falownika predkosc
      L     PIW [#Adres_1];	//zaladuj stw
      T     #STW;	//Slowo statusu
      T     #Slowo_Statusu;	//LW8
NETWORK
TITLE =
//Tworzenie slowa kontrolnego
// (network holds code this reader does not know; not shown)
//*********************************Blad Falownika
//*********************************Falownik gotowy do pracy
//**********************************Odblokuj falownik
//*********************************E-Stop Falownika
//*********************************Stop Falownika
//*********************************Start Falownika
//**
//      A     "Zawsze_False"
//*********************************Zaden z powyzszych warunkow
NETWORK
TITLE =
//Odczyt predkosc z falownika oraz  przypisanie predkosci od falownika.
//Zakres prekosci falownika:
//+-480HZ=+-24000
//
//1Hz=50 jednostek(dokladnosc 0.1Hz+pó³ cyfry)
//Predkosc bedzie zaokraglona do jednego miejsca po przecinku
//
//Predkosc zadana (zaokraglona z real do int)
//********************************Zadanie predkosci
pre1: L     #Predkosc_Zadana;	//50
      L     2.000000e+00;	//2
      /R;	//25
      L     1.000000e+02;
      *R;
      A     #Start_Prawo;
      JCN   e1;
      L     -1.000000e+00;
      *R;
e1:   RND;
pre2: T     #H_Temp;
      L     #H_Temp;
      T     PQW [#Adres_2];	//Transfer predkosci
//********************************Odczyt predkosci
//********************************
      L     #Timmer_Pom_2;
      T     #Timmer_Name;
      L     PIW [#Adres_2];
      ITD;
      DTR;
      L     2.000000e+00;
      *R;
      L     1.000000e+02;
      /R;
      T     #Predkosc_zwracana;	//predkosc odczytna z falownika
      L     0;
      ==R;
      L     S5T#2S300MS;
      SD    T [#Timmer_Name];
      A     T [#Timmer_Name];
      R     #Hamulec;
// BEU   
NETWORK
TITLE =
END_FUNCTION

FUNCTION "Zasprzeglenie_Bandy" : VOID	// FC 30
//Funkcja Zasprzeglajaca bande transportowa. Silnik lewo to kierunke przod
//
VERSION : 0.1
BEGIN
NETWORK
TITLE =
//Ten Network celowo jest wolny
//
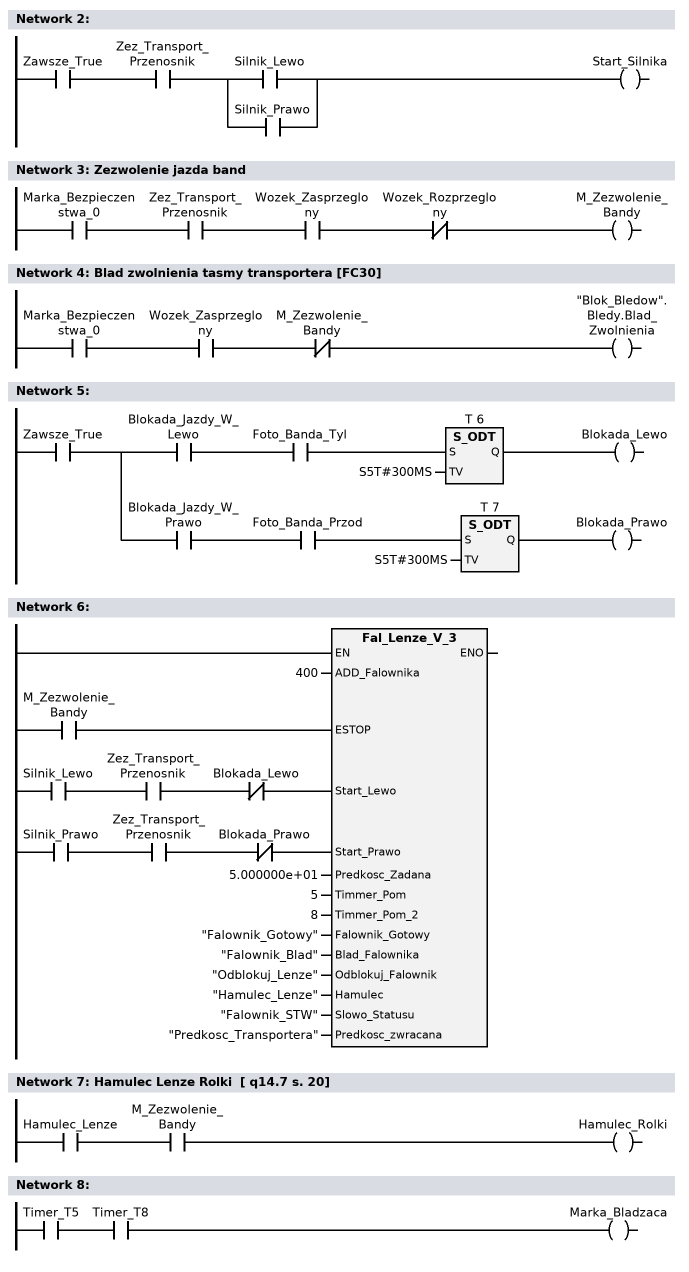
NETWORK
TITLE =
      A     "Zawsze_True";
      A     "Zez_Transport_Przenosnik";
      A(;
      O     "Silnik_Lewo";
      O     "Silnik_Prawo";
      );
      =     "Start_Silnika";
NETWORK
TITLE = Zezwolenie jazda band
//Zezwolenie na jazde band
//
      A     "Marka_Bezpieczenstwa_0";
      A     "Zez_Transport_Przenosnik";
      A     "Wozek_Zasprzeglony";
      AN    "Wozek_Rozprzeglony";
      =     "M_Zezwolenie_Bandy";
NETWORK
TITLE = Blad zwolnienia tasmy transportera [FC30]
//Blad zwolnienia transportera
      A     "Marka_Bezpieczenstwa_0";
      A     "Wozek_Zasprzeglony";
      AN    "M_Zezwolenie_Bandy";
      =     "Blok_Bledow".Bledy.Blad_Zwolnienia;
NETWORK
TITLE =
//blokada sinika w prawo
      A     "Zawsze_True";
      =     L 0.0;
      A     L 0.0;
      A     "Blokada_Jazdy_W_Lewo";
      A     "Foto_Banda_Tyl";
      L     S5T#300MS;
      SD    T 6;
      NOP   0;
      NOP   0;
      NOP   0;
      A     T 6;
      =     "Blokada_Lewo";
      A     L 0.0;
      A     "Blokada_Jazdy_W_Prawo";
      A     "Foto_Banda_Przod";
      L     S5T#300MS;
      SD    T 7;
      NOP   0;
      NOP   0;
      NOP   0;
      A     T 7;
      =     "Blokada_Prawo";
NETWORK
TITLE =
//Funkcja sterujaca falownikiem lenze
//
      A     "M_Zezwolenie_Bandy";
      =     L 0.0;
      BLD   103;
      A     "Silnik_Lewo";
      A     "Zez_Transport_Przenosnik";
      AN    "Blokada_Lewo";
      =     L 0.1;
      BLD   103;
      A     "Silnik_Prawo";
      A     "Zez_Transport_Przenosnik";
      AN    "Blokada_Prawo";
      =     L 0.2;
      BLD   103;
      CALL  "Fal_Lenze_V_3" (
           ADD_Falownika            := 400,
           ESTOP                    := L 0.0,
           Start_Lewo               := L 0.1,
           Start_Prawo              := L 0.2,
           Predkosc_Zadana          := 5.000000e+01,
           Timmer_Pom               := 5,
           Timmer_Pom_2             := 8,
           Falownik_Gotowy          := "Falownik_Gotowy",
           Blad_Falownika           := "Falownik_Blad",
           Odblokuj_Falownik        := "Odblokuj_Lenze",
           Hamulec                  := "Hamulec_Lenze",
           Slowo_Statusu            := "Falownik_STW",
           Predkosc_zwracana        := "Predkosc_Transportera");
      NOP   0;
NETWORK
TITLE = Hamulec Lenze Rolki  [ q14.7 s. 20]
      A     "Hamulec_Lenze";
      A     "M_Zezwolenie_Bandy";
      =     "Hamulec_Rolki";
NETWORK
TITLE =
//Sprawdzenie Timmera 
//
      A     "Timer_T5";
      A     "Timer_T8";
      =     "Marka_Bladzaca";
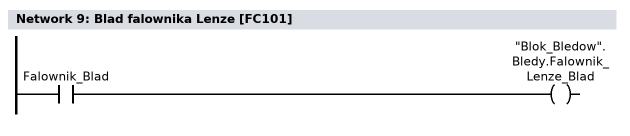
NETWORK
TITLE = Blad falownika Lenze [FC101]
      A     "Falownik_Blad";
      =     "Blok_Bledow".Bledy.Falownik_Lenze_Blad;
END_FUNCTION

FUNCTION "Odbieranie_Danych" : VOID	// FC 41
VERSION : 0.1
VAR_INPUT
  i_Zad_Transmisji_0_0 : BOOL ;
  i_Zad_Danych_0_1 : BOOL ;
  io_Toggle_0_2 : BOOL ;
  i_0_3 : BOOL ;
  i_0_4 : BOOL ;
  i_Funkcja_Receive_0_5 : BOOL ;
  i_Funkcja_Share_0_6 : BOOL ;
  i_0_7 : BOOL ;
  ib_1_0 : BYTE ;
  iw_Nr_Bloku_2_0 : INT ;
  iw_Kanal_Odbioru_4_0 : WORD ;
  iow_Licz_Rekordow_6_0 : INT ;
END_VAR
VAR_OUTPUT
  M_i_Zad_Transmisji_0_0 : BOOL ;
  M_i_Zad_Danych_0_1 : BOOL ;
  M_io_Toggle_0_2 : BOOL ;
  M_i_Funkcja_Receive_0_3 : BOOL ;
  M_i_Funkcja_Share_0_4 : BOOL ;
  M_i_0_5 : BOOL ;
  M_i_0_6 : BOOL ;
  M_i_0_7 : BOOL ;
  M_ib_1_0 : BYTE ;
  M_iw_Nr_Bloku_2_0 : INT ;
  M_iw_Kanal_Odbioru_4_0 : WORD ;
  M_iow_Licz_Rekordow_6_0 : INT ;
END_VAR
BEGIN
NETWORK
TITLE =
//Ten Network celowo jest wolny
NETWORK
TITLE =
//Przypisanie do wyjsc
      A     #i_Zad_Transmisji_0_0;
      =     #M_i_Zad_Transmisji_0_0;
      A     #i_Zad_Danych_0_1;
      =     #M_i_Zad_Danych_0_1;
      A     #io_Toggle_0_2;
      =     #M_io_Toggle_0_2;
      A     #i_Funkcja_Receive_0_5;
      =     #M_i_Funkcja_Receive_0_3;
      A     #i_Funkcja_Share_0_6;
      =     #M_i_Funkcja_Share_0_4;
      A     #i_0_3;
      =     #M_i_0_5;
      A     #i_0_4;
      =     #M_i_0_6;
      A     #i_0_7;
      =     #M_i_0_7;
      L     #ib_1_0;
      T     #M_ib_1_0;
      L     #iw_Nr_Bloku_2_0;
      T     #M_iw_Nr_Bloku_2_0;
      L     #iw_Kanal_Odbioru_4_0;
      T     #M_iw_Kanal_Odbioru_4_0;
      L     #iow_Licz_Rekordow_6_0;
      T     #M_iow_Licz_Rekordow_6_0;
END_FUNCTION

FUNCTION "Wysylanie_Danych" : VOID	// FC 42
VERSION : 0.1
VAR_INPUT
  M_o_Trans_Ustawiona_0_0 : BOOL ;
  M_o_Blok_Zarez_0_1 : BOOL ;
  M_oi_Toggle_0_2 : BOOL ;
  M_o_Przesyl_Danych_0_3 : BOOL ;
  M_o_Koniec_Nadawania_0_4 : BOOL ;
  M_o_F_Receive_Wybr_0_5 : BOOL ;
  M_o_F_Share_Wybr_0_6 : BOOL ;
  M_o_0_7 : BOOL ;
  M_ob_1_0_1 : BYTE ;
  M_ow_Nr_Rekordu_2_0 : INT ;
  M_ow_Kan_Pobierania_4_0 : WORD ;
  M_oiw_Licz_Rekordu_6_0 : INT ;
END_VAR
VAR_OUTPUT
  o_Trans_Ustawiona_0_0 : BOOL ;
  o_Blok_Zarez_0_1 : BOOL ;
  oi_Toggle_0_2 : BOOL ;
  o_Przesyl_Danych_0_3 : BOOL ;
  o_Koniec_Nadawania_0_4 : BOOL ;
  o_F_Receive_Wybr_0_5 : BOOL ;
  o_F_Share_Wybr_0_6 : BOOL ;
  o_0_7 : BOOL ;
  ob_1_0 : BYTE ;
  ow_Nr_Rekordu_2_0 : INT ;
  ow_Kanal_Pobierania_4_0 : WORD ;
  oiw_Licznik_Rekordu_6_0 : INT ;
END_VAR
BEGIN
NETWORK
TITLE =
//Ten Network celowo jest wolny
NETWORK
TITLE =
      A     #M_o_Trans_Ustawiona_0_0;
      =     #o_Trans_Ustawiona_0_0;
      A     #M_o_Blok_Zarez_0_1;
      =     #o_Blok_Zarez_0_1;
      A     #M_o_Przesyl_Danych_0_3;
      =     #o_Przesyl_Danych_0_3;
      A     #M_o_Koniec_Nadawania_0_4;
      =     #o_Koniec_Nadawania_0_4;
      A     #M_oi_Toggle_0_2;
      =     #oi_Toggle_0_2;
      A     #M_o_F_Receive_Wybr_0_5;
      =     #o_F_Receive_Wybr_0_5;
      A     #M_o_F_Share_Wybr_0_6;
      =     #o_F_Share_Wybr_0_6;
      A     #M_o_0_7;
      =     #o_0_7;
      L     #M_ob_1_0_1;
      T     #ob_1_0;
      L     #M_ow_Nr_Rekordu_2_0;
      T     #ow_Nr_Rekordu_2_0;
      L     #M_ow_Kan_Pobierania_4_0;
      T     #ow_Kanal_Pobierania_4_0;
      L     #M_oiw_Licz_Rekordu_6_0;
      T     #oiw_Licznik_Rekordu_6_0;
END_FUNCTION

FUNCTION "Aufruf Achse 1" : VOID	// FC 100
TITLE = Aufruf Achse 1 (Adresse 256)
//Dieses Programmbeispiel zeigt nur die prinzipielle Vorgehensweise.
//Für fehlerhafte Programmfunktionen und deren Folgen
//kann weder eine juristische, noch irgendeine Haftung übernommen werden!
VERSION : 0.1
BEGIN
NETWORK
TITLE = Ansteuerung Achse_1 (Adr. 256)
//Die FC140 dient als Beispielprogrammbaustein zur Ansteuerung des 
//Applikationsmoduls "Erweiterte Buspositionierung" für die Gerätereihen 
//MOVIDRIVE in Technologieausführung.
//
//Mit Hilfe der FC140 können die Antriebsumrichter via PROFIBUS DP oder PROFINET 
//I/O angesteuert werden.
//
//Nach einer Inbetriebnahme des Applikationsmoduls können die Prozeßdaten im 
//Monitor der Buspositionierung visualisiert werden. Weitere Informationen wie 
//z.B. die Kodierung der Prozeßdaten sind in der Onlinehilfe der MOVITOOLS 
//dokumentiert.
//
//Eingänge der FC:
//"DRIVE_IO_ADDRESS": Anfangsadresse des E/A-Bereichs => Hardwarekonfiguration
//"ENABLE_RAPID_STOP" = true: Freigabe; false: Schnellstopp
//"RESET": Fehler quittieren
//Die Betriebsart wird mit den Eingängen "Jog_plus_mode, Jog_minus_mode; 
//Ref_travel und Positioning_mode angewählt.
//"SETPOINT_POS": Positionssollwert (DINT) in Anwendereinheit.
//Die Anwendereinheit ist abhängig von der Inbetriebnahme der "Erweiterten 
//Buspositionierung"
//"SETPOINT_SPEED": Positioniergeschwindigkeit (INT) in rpm
//"START_RAMP": Beschleunigungsrampe (INT) in ms
//"STOP_RAMP": Verzögerungsrampe(INT) in ms
//
//Ausgänge der FC"
//Ist die Datenübertragung/PROFIBUS gestört, so werden alle Ausgänge abgelöscht.
//=> "COMMUNICATION_OK = false (selbstquittierend)
//"FAULT_OF_AXIS" = true: Ein Fehler steht an.
//"WARNING_OF_AXIS" = true: Eine Warnung steht an.
//"INVERTER_READY" = true: Es liegt kein Fehler vor & Netzspannung EIN"
//"REFERENCED" = true: Die Achse ist referenziert
//TARGET_POS_REACHED" = true: Die Zielposition ist erreicht.
//"AXIS_INTERLOCKED" = true: Meldet zurück, daß eine unplausible Modeanwahl 
//vorliegt. (=> keine oder mehrere Modi angewählt)
//"FAULT_NO" <> 0: Die Fehlercodes sind im Systemhandbuch dokumentiert und werden 
//in den MOVITOOLS (Status, Busmonitor) angezeigt.
//"ACTUAL_POSITION": Positionsistwert (DINT) in Anwendereinheit.
//"ACTUAL_SPEED": Istgeschwindigkeit (INT) in rpm
//"ACTUAL_CURRENT": Stromistwert (Wirkstrom) in Prozent vom Gerätenennstrom
//
//
//Hinweis: Endschalter freifahren (F27):
//Ist ein Endschalter angefahren, so wird die Achse mit Notstopp stillgesetzt 
//und F27 gemeldet. Wählen Sie Reset und richtungsabhängig Tippen_plus bzw. 
//Tippen_minus an. Der Antrieb wird dadurch automatisch mit der Motordrehzahl n = 
//100 1/min freigefahren.
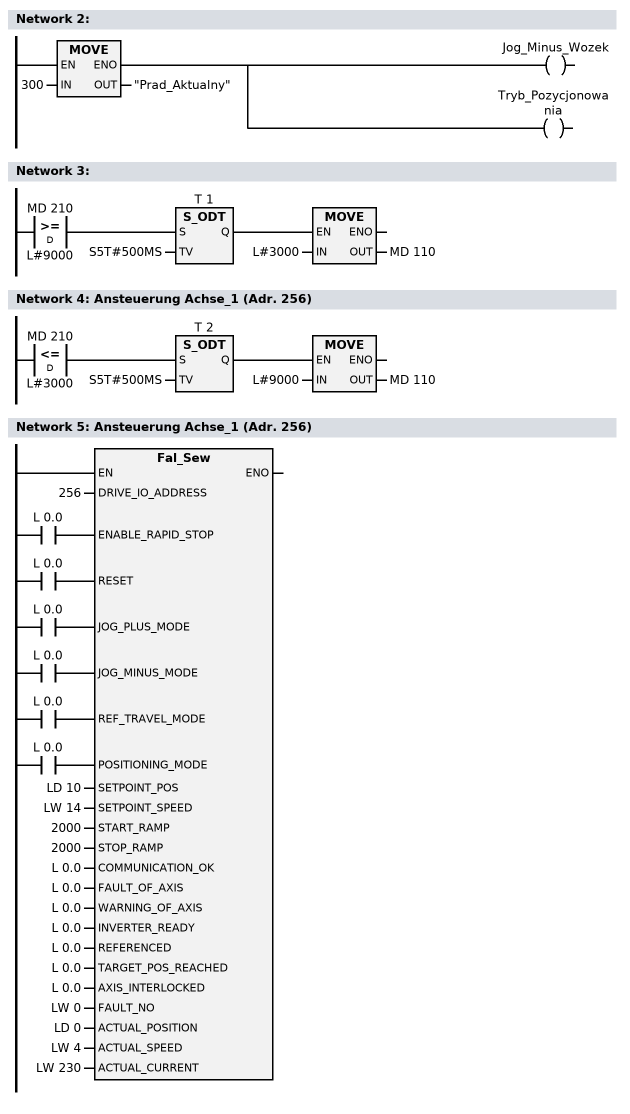
NETWORK
TITLE =
      L     300;
      T     "Prad_Aktualny";
      SET;
      SAVE;
      CLR;
      A     BR;
      =     "Jog_Minus_Wozek";
      =     "Tryb_Pozycjonowania";
NETWORK
TITLE =
      A(;
      A(;
      L     MD 210;
      L     L#9000;
      >=D;
      );
      L     S5T#500MS;
      SD    T 1;
      NOP   0;
      NOP   0;
      NOP   0;
      A     T 1;
      );
      JNB   _001;
      L     L#3000;
      T     MD 110;
_001: NOP   0;
NETWORK
TITLE = Ansteuerung Achse_1 (Adr. 256)
      A(;
      A(;
      L     MD 210;
      L     L#3000;
      <=D;
      );
      L     S5T#500MS;
      SD    T 2;
      NOP   0;
      NOP   0;
      NOP   0;
      A     T 2;
      );
      JNB   _002;
      L     L#9000;
      T     MD 110;
_002: NOP   0;
NETWORK
TITLE = Ansteuerung Achse_1 (Adr. 256)
      A     L 0.0;
      =     L 232.0;
      BLD   103;
      A     L 0.0;
      =     L 232.1;
      BLD   103;
      A     L 0.0;
      =     L 232.2;
      BLD   103;
      A     L 0.0;
      =     L 232.3;
      BLD   103;
      A     L 0.0;
      =     L 232.4;
      BLD   103;
      A     L 0.0;
      =     L 232.5;
      BLD   103;
      CALL  "Fal_Sew" (
           DRIVE_IO_ADDRESS         := 256,
           ENABLE_RAPID_STOP        := L 232.0,
           RESET                    := L 232.1,
           JOG_PLUS_MODE            := L 232.2,
           JOG_MINUS_MODE           := L 232.3,
           REF_TRAVEL_MODE          := L 232.4,
           POSITIONING_MODE         := L 232.5,
           SETPOINT_POS             := LD 10,
           SETPOINT_SPEED           := LW 14,
           START_RAMP               := 2000,
           STOP_RAMP                := 2000,
           COMMUNICATION_OK         := L 0.0,
           FAULT_OF_AXIS            := L 0.0,
           WARNING_OF_AXIS          := L 0.0,
           INVERTER_READY           := L 0.0,
           REFERENCED               := L 0.0,
           TARGET_POS_REACHED       := L 0.0,
           AXIS_INTERLOCKED         := L 0.0,
           FAULT_NO                 := LW 0,
           ACTUAL_POSITION          := LD 0,
           ACTUAL_SPEED             := LW 4,
           ACTUAL_CURRENT           := LW 230);
      NOP   0;
END_FUNCTION

FUNCTION "Jazda_Shuttle" : VOID	// FC 101
//Funkcja odpowiada za jazde Shuttle na pozycje. Funkcja pobrana ze stron SEW.
VERSION : 0.1
BEGIN
NETWORK
TITLE = Ansteuerung Achse_1 (Adr. 256)
//Die FC140 dient als Beispielprogrammbaustein zur Ansteuerung des 
//Applikationsmoduls "Erweiterte Buspositionierung" für die Gerätereihen 
//MOVIDRIVE in Technologieausführung.
//
//Mit Hilfe der FC140 können die Antriebsumrichter via PROFIBUS DP oder PROFINET 
//I/O angesteuert werden.
//
//Nach einer Inbetriebnahme des Applikationsmoduls können die Prozeßdaten im 
//Monitor der Buspositionierung visualisiert werden. Weitere Informationen wie 
//z.B. die Kodierung der Prozeßdaten sind in der Onlinehilfe der MOVITOOLS 
//dokumentiert.
//
//Eingänge der FC:
//"DRIVE_IO_ADDRESS": Anfangsadresse des E/A-Bereichs => Hardwarekonfiguration
//"ENABLE_RAPID_STOP" = true: Freigabe; false: Schnellstopp
//"RESET": Fehler quittieren
//Die Betriebsart wird mit den Eingängen "Jog_plus_mode, Jog_minus_mode; 
//Ref_travel und Positioning_mode angewählt.
//"SETPOINT_POS": Positionssollwert (DINT) in Anwendereinheit.
//Die Anwendereinheit ist abhängig von der Inbetriebnahme der "Erweiterten 
//Buspositionierung"
//"SETPOINT_SPEED": Positioniergeschwindigkeit (INT) in rpm
//"START_RAMP": Beschleunigungsrampe (INT) in ms
//"STOP_RAMP": Verzögerungsrampe(INT) in ms
//
//Ausgänge der FC"
//Ist die Datenübertragung/PROFIBUS gestört, so werden alle Ausgänge abgelöscht.
//=> "COMMUNICATION_OK = false (selbstquittierend)
//"FAULT_OF_AXIS" = true: Ein Fehler steht an.
//"WARNING_OF_AXIS" = true: Eine Warnung steht an.
//"INVERTER_READY" = true: Es liegt kein Fehler vor & Netzspannung EIN"
//"REFERENCED" = true: Die Achse ist referenziert
//TARGET_POS_REACHED" = true: Die Zielposition ist erreicht.
//"AXIS_INTERLOCKED" = true: Meldet zurück, daß eine unplausible Modeanwahl 
//vorliegt. (=> keine oder mehrere Modi angewählt)
//"FAULT_NO" <> 0: Die Fehlercodes sind im Systemhandbuch dokumentiert und werden 
//in den MOVITOOLS (Status, Busmonitor) angezeigt.
//"ACTUAL_POSITION": Positionsistwert (DINT) in Anwendereinheit.
//"ACTUAL_SPEED": Istgeschwindigkeit (INT) in rpm
//"ACTUAL_CURRENT": Stromistwert (Wirkstrom) in Prozent vom Gerätenennstrom
//
//
//Hinweis: Endschalter freifahren (F27):
//Ist ein Endschalter angefahren, so wird die Achse mit Notstopp stillgesetzt 
//und F27 gemeldet. Wählen Sie Reset und richtungsabhängig Tippen_plus bzw. 
//Tippen_minus an. Der Antrieb wird dadurch automatisch mit der Motordrehzahl n = 
//100 1/min freigefahren.
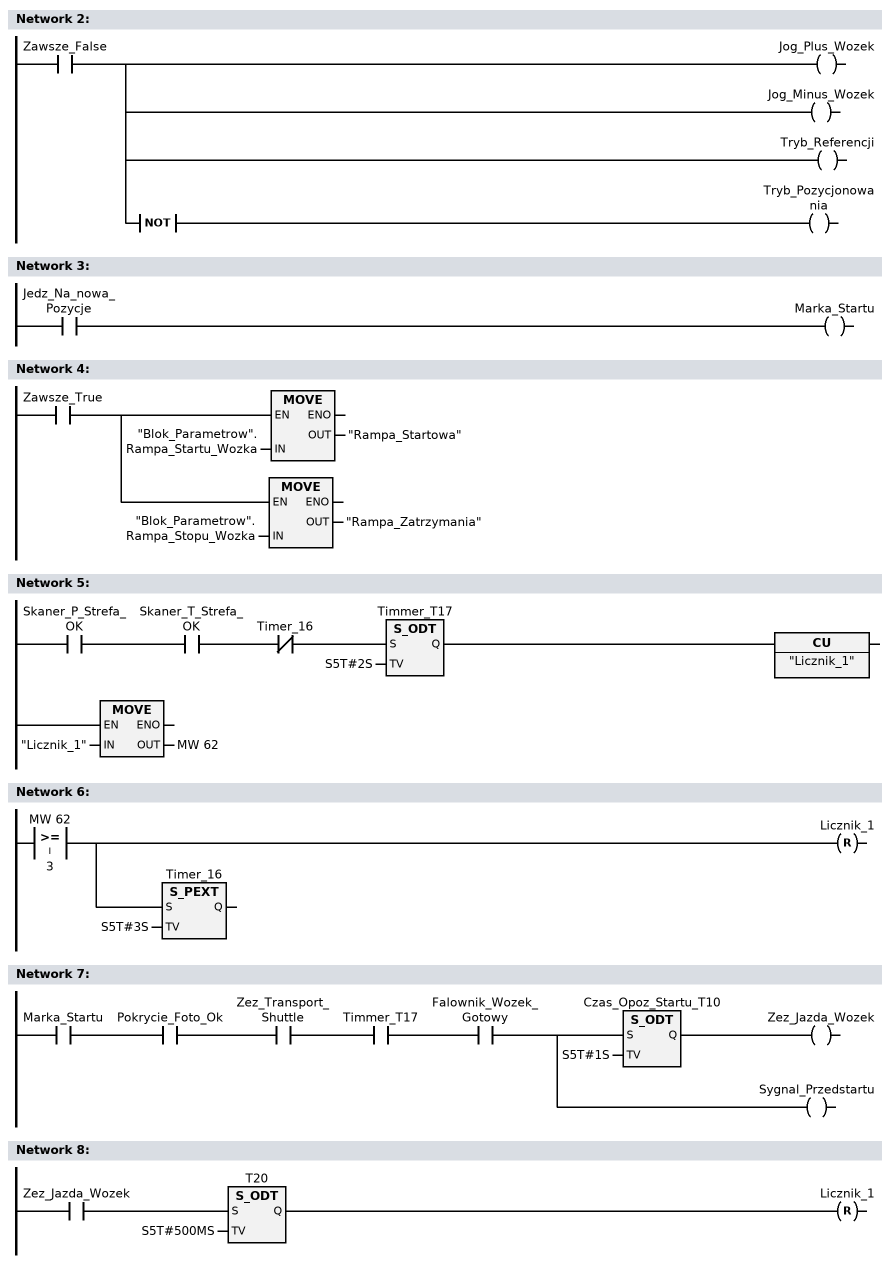
NETWORK
TITLE =
//Wyzerowanie odpowiednich bitow
      A     "Zawsze_False";
      =     L 0.0;
      A     L 0.0;
      BLD   102;
      =     "Jog_Plus_Wozek";
      A     L 0.0;
      BLD   102;
      =     "Jog_Minus_Wozek";
      A     L 0.0;
      BLD   102;
      =     "Tryb_Referencji";
      A     L 0.0;
      NOT;
      =     "Tryb_Pozycjonowania";
NETWORK
TITLE =
//Tryb pozycjonowania
//      A     "Zawsze_True"
//      =     "Tryb_Pozycjonowania"
//
      A     "Jedz_Na_nowa_Pozycje";
      =     "Marka_Startu";
NETWORK
TITLE =
//Przepisanie wartosci ramp
      A     "Zawsze_True";
      =     L 0.0;
      A     L 0.0;
      JNB   _001;
      L     "Blok_Parametrow".Rampa_Startu_Wozka;
      T     "Rampa_Startowa";
_001: NOP   0;
      A     L 0.0;
      JNB   _002;
      L     "Blok_Parametrow".Rampa_Stopu_Wozka;
      T     "Rampa_Zatrzymania";
_002: NOP   0;
NETWORK
TITLE =
      A(;
      A     "Skaner_P_Strefa_OK";
      A     "Skaner_T_Strefa_OK";
      AN    "Timer_16";
      L     S5T#2S;
      SD    "Timmer_T17";
      NOP   0;
      NOP   0;
      NOP   0;
      A     "Timmer_T17";
      );
      CU    "Licznik_1";
      BLD   101;
      NOP   0;
      NOP   0;
      NOP   0;
      L     "Licznik_1";
      T     MW 62;
      NOP   0;
      NOP   0;
NETWORK
TITLE =
//Podlicz jak trzy bledy to czekaj 5s
//
      L     MW 62;
      L     3;
      >=I;
      =     L 0.0;
      A     L 0.0;
      BLD   102;
      R     "Licznik_1";
      A     L 0.0;
      L     S5T#3S;
      SE    "Timer_16";
      NOP   0;
      NOP   0;
      NOP   0;
      NOP   0;
NETWORK
TITLE =
//Pokrycie foto bezpieczne
      A     "Marka_Startu";
      A     "Pokrycie_Foto_Ok";
      A     "Zez_Transport_Shuttle";
      A     "Timmer_T17";
      A     "Falownik_Wozek_Gotowy";
      =     L 0.0;
      A     L 0.0;
      L     S5T#1S;
      SD    "Czas_Opoz_Startu_T10";
      NOP   0;
      NOP   0;
      NOP   0;
      A     "Czas_Opoz_Startu_T10";
      =     "Zez_Jazda_Wozek";
      A     L 0.0;
      BLD   102;
      =     "Sygnal_Przedstartu";
NETWORK
TITLE =
      A     "Zez_Jazda_Wozek";
      L     S5T#500MS;
      SD    "T20";
      NOP   0;
      NOP   0;
      NOP   0;
      A     "T20";
      R     "Licznik_1";
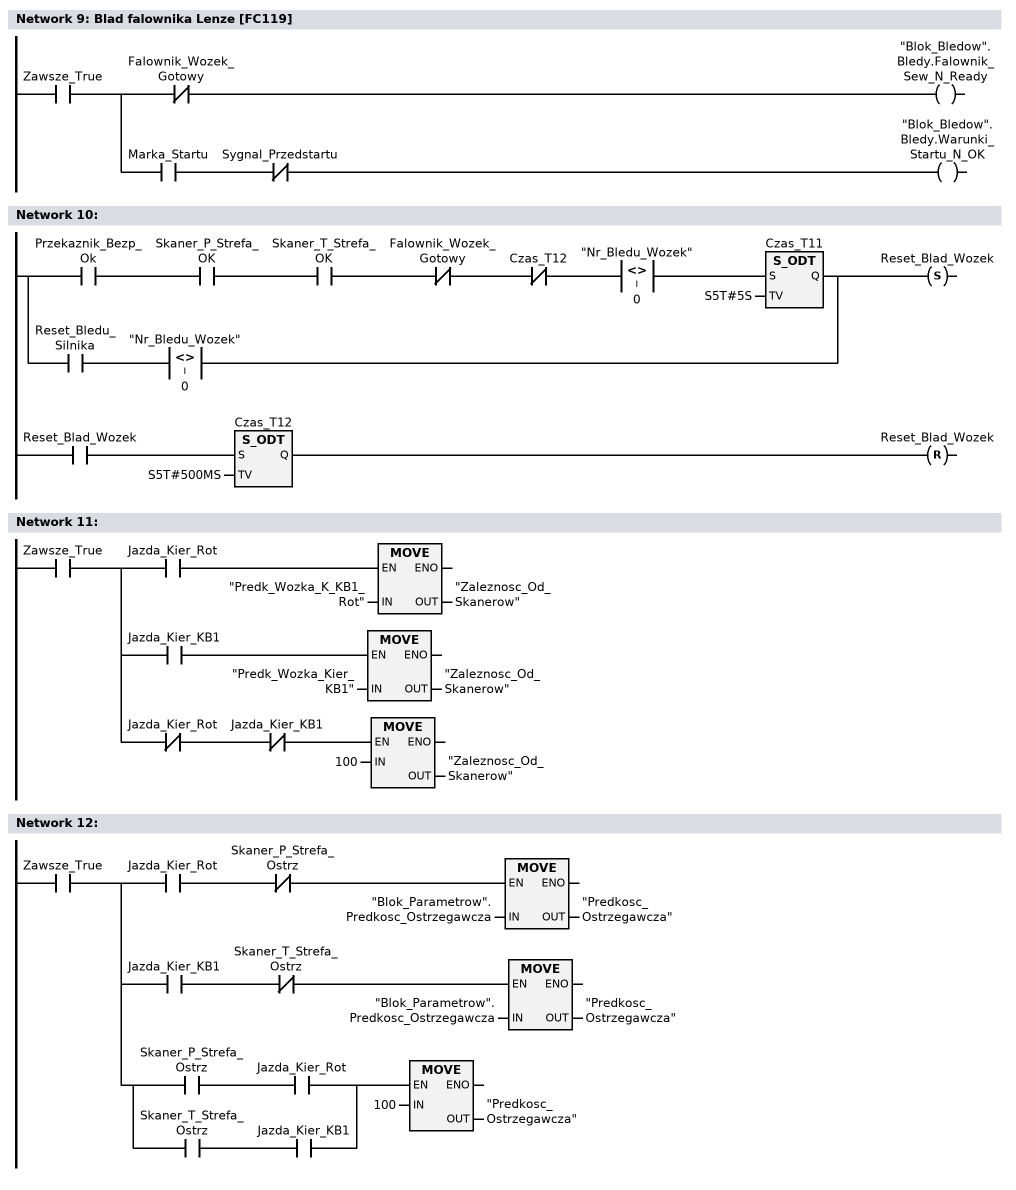
NETWORK
TITLE = Blad falownika Lenze [FC119]
//Falownik sew nie gotowy
      A     "Zawsze_True";
      =     L 0.0;
      A     L 0.0;
      AN    "Falownik_Wozek_Gotowy";
      =     "Blok_Bledow".Bledy.Falownik_Sew_N_Ready;
      A     L 0.0;
      A     "Marka_Startu";
      AN    "Sygnal_Przedstartu";
      =     "Blok_Bledow".Bledy.Warunki_Startu_N_OK;
NETWORK
TITLE =
//Funkcja autoresetu silnika jazdy wozka
      A(;
      O(;
      A     "Przekaznik_Bezp_Ok";
      A     "Skaner_P_Strefa_OK";
      A     "Skaner_T_Strefa_OK";
      AN    "Falownik_Wozek_Gotowy";
      AN    "Czas_T12";
      A(;
      L     "Nr_Bledu_Wozek";
      L     0;
      <>I;
      );
      L     S5T#5S;
      SD    "Czas_T11";
      NOP   0;
      NOP   0;
      NOP   0;
      A     "Czas_T11";
      );
      O;
      A     "Reset_Bledu_Silnika";
      A(;
      L     "Nr_Bledu_Wozek";
      L     0;
      <>I;
      );
      );
      S     "Reset_Blad_Wozek";
      A(;
      A     "Reset_Blad_Wozek";
      L     S5T#500MS;
      SD    "Czas_T12";
      NOP   0;
      NOP   0;
      NOP   0;
      A     "Czas_T12";
      );
      R     "Reset_Blad_Wozek";
      NOP   0;
NETWORK
TITLE =
//Zmiana predosc na podstawie polozenia
      A     "Zawsze_True";
      =     L 0.0;
      A     L 0.0;
      A     "Jazda_Kier_Rot";
      JNB   _003;
      L     "Predk_Wozka_K_KB1_Rot";
      T     "Zaleznosc_Od_Skanerow";
_003: NOP   0;
      A     L 0.0;
      A     "Jazda_Kier_KB1";
      JNB   _004;
      L     "Predk_Wozka_Kier_KB1";
      T     "Zaleznosc_Od_Skanerow";
_004: NOP   0;
      A     L 0.0;
      AN    "Jazda_Kier_Rot";
      AN    "Jazda_Kier_KB1";
      JNB   _005;
      L     100;
      T     "Zaleznosc_Od_Skanerow";
_005: NOP   0;
NETWORK
TITLE =
//Zmiana predkosci po wejsiu w warnning
      A     "Zawsze_True";
      =     L 0.0;
      A     L 0.0;
      A     "Jazda_Kier_Rot";
      AN    "Skaner_P_Strefa_Ostrz";
      JNB   _006;
      L     "Blok_Parametrow".Predkosc_Ostrzegawcza;
      T     "Predkosc_Ostrzegawcza";
_006: NOP   0;
      A     L 0.0;
      A     "Jazda_Kier_KB1";
      AN    "Skaner_T_Strefa_Ostrz";
      JNB   _007;
      L     "Blok_Parametrow".Predkosc_Ostrzegawcza;
      T     "Predkosc_Ostrzegawcza";
_007: NOP   0;
      A     L 0.0;
      A(;
      A     "Skaner_P_Strefa_Ostrz";
      A     "Jazda_Kier_Rot";
      O;
      A     "Skaner_T_Strefa_Ostrz";
      A     "Jazda_Kier_KB1";
      );
      JNB   _008;
      L     100;
      T     "Predkosc_Ostrzegawcza";
_008: NOP   0;
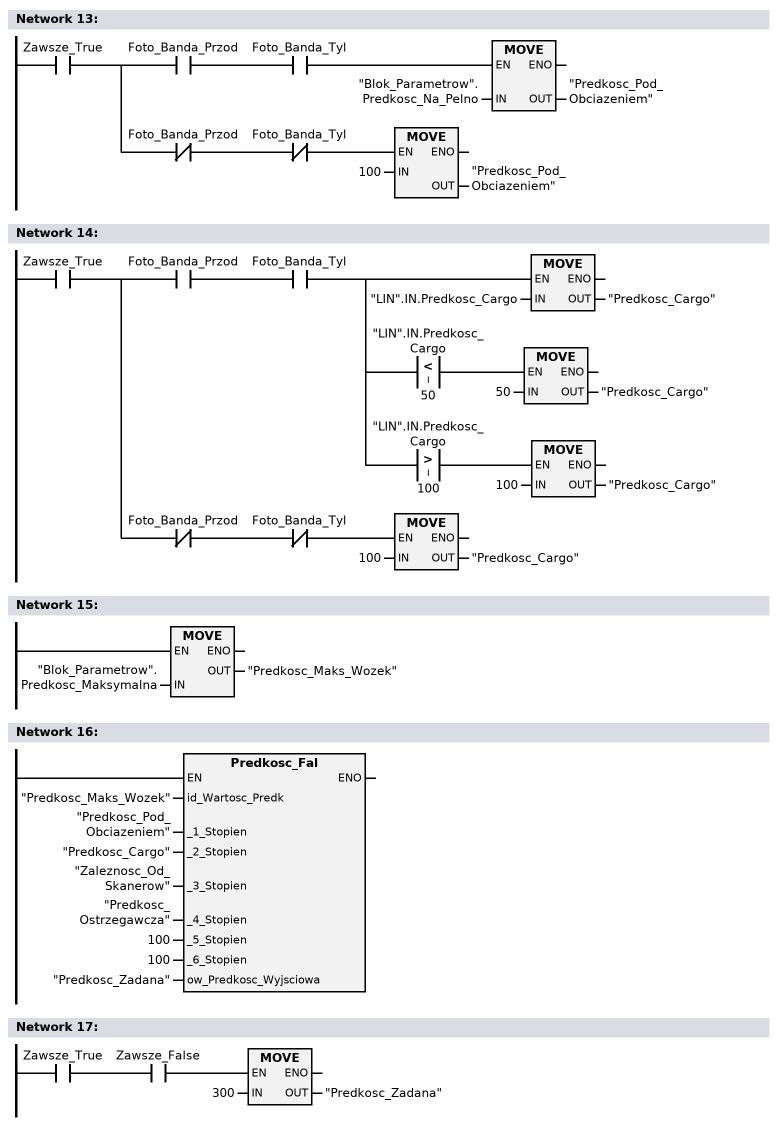
NETWORK
TITLE =
//Zmiana prdkosci gdy na pusto lub pelno
      A     "Zawsze_True";
      =     L 0.0;
      A     L 0.0;
      A     "Foto_Banda_Przod";
      A     "Foto_Banda_Tyl";
      JNB   _009;
      L     "Blok_Parametrow".Predkosc_Na_Pelno;
      T     "Predkosc_Pod_Obciazeniem";
_009: NOP   0;
      A     L 0.0;
      AN    "Foto_Banda_Przod";
      AN    "Foto_Banda_Tyl";
      JNB   _00a;
      L     100;
      T     "Predkosc_Pod_Obciazeniem";
_00a: NOP   0;
NETWORK
TITLE =
//Predkosc po uwzglednieniu funkcji cargo. Zakres predkosci cargo to  wartosci 50 
//do 100%
      A     "Zawsze_True";
      =     L 0.0;
      A     L 0.0;
      A     "Foto_Banda_Przod";
      A     "Foto_Banda_Tyl";
      =     L 0.1;
      A     L 0.1;
      JNB   _00b;
      L     "LIN".IN.Predkosc_Cargo;
      T     "Predkosc_Cargo";
_00b: NOP   0;
      A     L 0.1;
      A(;
      L     "LIN".IN.Predkosc_Cargo;
      L     50;
      <I;
      );
      JNB   _00c;
      L     50;
      T     "Predkosc_Cargo";
_00c: NOP   0;
      A     L 0.1;
      A(;
      L     "LIN".IN.Predkosc_Cargo;
      L     100;
      >I;
      );
      JNB   _00d;
      L     100;
      T     "Predkosc_Cargo";
_00d: NOP   0;
      A     L 0.0;
      AN    "Foto_Banda_Przod";
      AN    "Foto_Banda_Tyl";
      JNB   _00e;
      L     100;
      T     "Predkosc_Cargo";
_00e: NOP   0;
NETWORK
TITLE =
      L     "Blok_Parametrow".Predkosc_Maksymalna;
      T     "Predkosc_Maks_Wozek";
      NOP   0;
NETWORK
TITLE =
      CALL  "Predkosc_Fal" (
           id_Wartosc_Predk         := "Predkosc_Maks_Wozek",
           _1_Stopien               := "Predkosc_Pod_Obciazeniem",
           _2_Stopien               := "Predkosc_Cargo",
           _3_Stopien               := "Zaleznosc_Od_Skanerow",
           _4_Stopien               := "Predkosc_Ostrzegawcza",
           _5_Stopien               := 100,
           _6_Stopien               := 100,
           ow_Predkosc_Wyjsciowa    := "Predkosc_Zadana");
      NOP   0;
NETWORK
TITLE =
      A     "Zawsze_True";
      A     "Zawsze_False";
      JNB   _00f;
      L     300;
      T     "Predkosc_Zadana";
_00f: NOP   0;
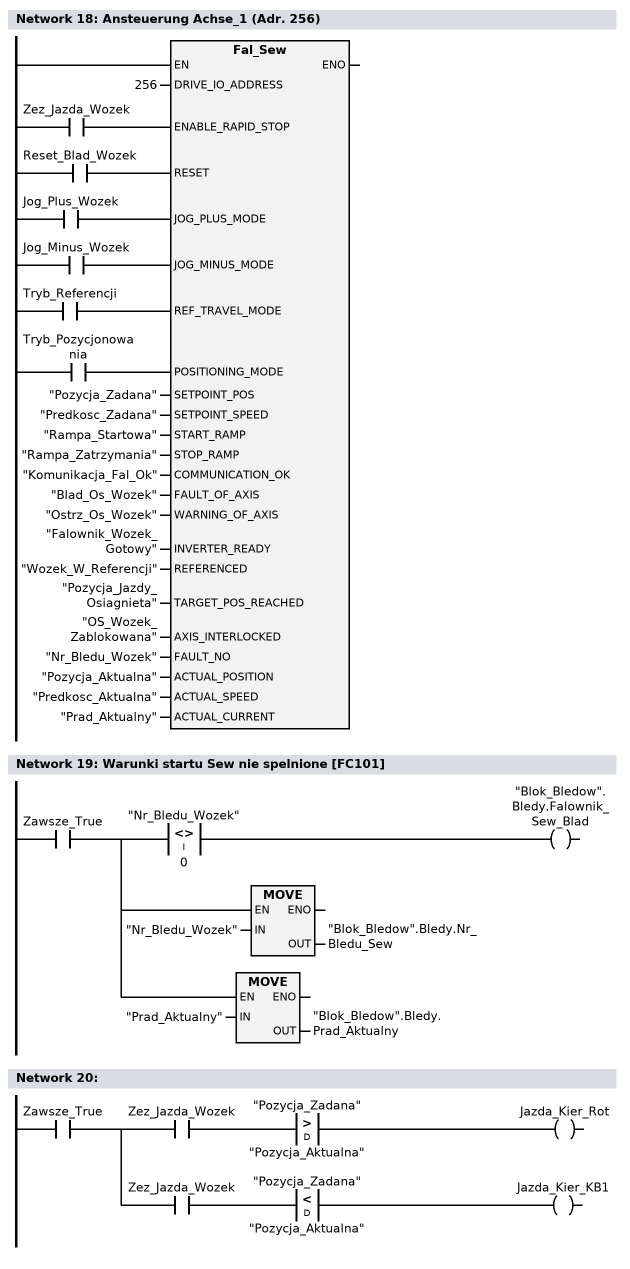
NETWORK
TITLE = Ansteuerung Achse_1 (Adr. 256)
//Warosc pozycji podawana jest mm
//Rampy sa w ms
      A     "Zez_Jazda_Wozek";
      =     L 0.0;
      BLD   103;
      A     "Reset_Blad_Wozek";
      =     L 0.1;
      BLD   103;
      A     "Jog_Plus_Wozek";
      =     L 0.2;
      BLD   103;
      A     "Jog_Minus_Wozek";
      =     L 0.3;
      BLD   103;
      A     "Tryb_Referencji";
      =     L 0.4;
      BLD   103;
      A     "Tryb_Pozycjonowania";
      =     L 0.5;
      BLD   103;
      CALL  "Fal_Sew" (
           DRIVE_IO_ADDRESS         := 256,
           ENABLE_RAPID_STOP        := L 0.0,
           RESET                    := L 0.1,
           JOG_PLUS_MODE            := L 0.2,
           JOG_MINUS_MODE           := L 0.3,
           REF_TRAVEL_MODE          := L 0.4,
           POSITIONING_MODE         := L 0.5,
           SETPOINT_POS             := "Pozycja_Zadana",
           SETPOINT_SPEED           := "Predkosc_Zadana",
           START_RAMP               := "Rampa_Startowa",
           STOP_RAMP                := "Rampa_Zatrzymania",
           COMMUNICATION_OK         := "Komunikacja_Fal_Ok",
           FAULT_OF_AXIS            := "Blad_Os_Wozek",
           WARNING_OF_AXIS          := "Ostrz_Os_Wozek",
           INVERTER_READY           := "Falownik_Wozek_Gotowy",
           REFERENCED               := "Wozek_W_Referencji",
           TARGET_POS_REACHED       := "Pozycja_Jazdy_Osiagnieta",
           AXIS_INTERLOCKED         := "OS_Wozek_Zablokowana",
           FAULT_NO                 := "Nr_Bledu_Wozek",
           ACTUAL_POSITION          := "Pozycja_Aktualna",
           ACTUAL_SPEED             := "Predkosc_Aktualna",
           ACTUAL_CURRENT           := "Prad_Aktualny");
      NOP   0;
NETWORK
TITLE = Warunki startu Sew nie spelnione [FC101]
//Blad falownika sew
      A     "Zawsze_True";
      =     L 0.0;
      A     L 0.0;
      A(;
      L     "Nr_Bledu_Wozek";
      L     0;
      <>I;
      );
      =     "Blok_Bledow".Bledy.Falownik_Sew_Blad;
      A     L 0.0;
      JNB   _010;
      L     "Nr_Bledu_Wozek";
      T     "Blok_Bledow".Bledy.Nr_Bledu_Sew;
_010: NOP   0;
      A     L 0.0;
      JNB   _011;
      L     "Prad_Aktualny";
      T     "Blok_Bledow".Bledy.Prad_Aktualny;
_011: NOP   0;
NETWORK
TITLE =
//Wyznaczenie kierunku jazdy
//kb1 3000
//
//kb2-12000
//
//
//rot-1000000000000
      A     "Zawsze_True";
      =     L 0.0;
      A     L 0.0;
      A     "Zez_Jazda_Wozek";
      A(;
      L     "Pozycja_Zadana";
      L     "Pozycja_Aktualna";
      >D;
      );
      =     "Jazda_Kier_Rot";
      A     L 0.0;
      A     "Zez_Jazda_Wozek";
      A(;
      L     "Pozycja_Zadana";
      L     "Pozycja_Aktualna";
      <D;
      );
      =     "Jazda_Kier_KB1";
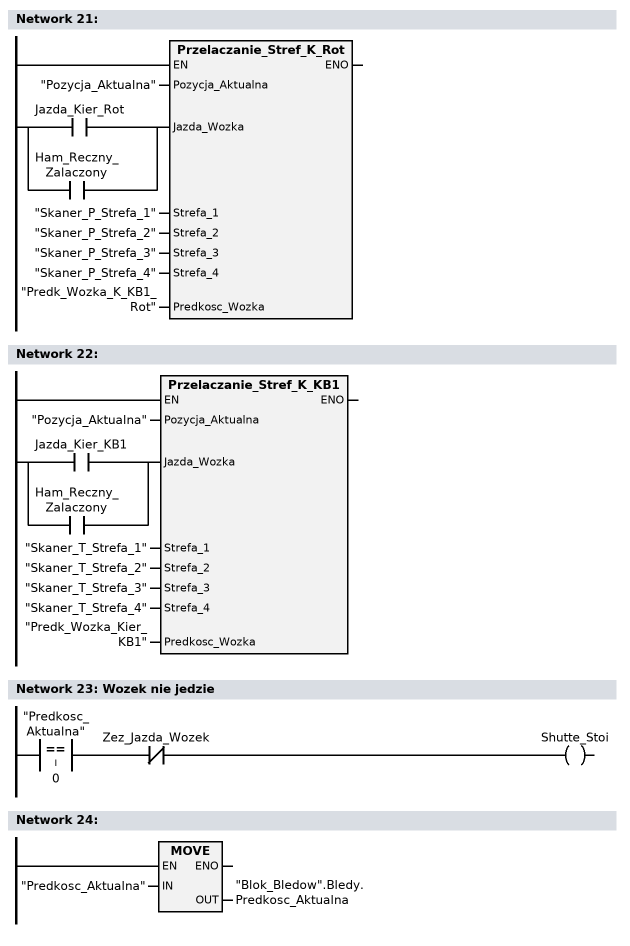
NETWORK
TITLE =
//Jazda w kierunku kb1-rotacja
//
      A(;
      O     "Jazda_Kier_Rot";
      O     "Ham_Reczny_Zalaczony";
      );
      =     L 0.0;
      BLD   103;
      CALL  "Przelaczanie_Stref_K_Rot" (
           Pozycja_Aktualna         := "Pozycja_Aktualna",
           Jazda_Wozka              := L 0.0,
           Strefa_1                 := "Skaner_P_Strefa_1",
           Strefa_2                 := "Skaner_P_Strefa_2",
           Strefa_3                 := "Skaner_P_Strefa_3",
           Strefa_4                 := "Skaner_P_Strefa_4",
           Predkosc_Wozka           := "Predk_Wozka_K_KB1_Rot");
      NOP   0;
NETWORK
TITLE =
      A(;
      O     "Jazda_Kier_KB1";
      O     "Ham_Reczny_Zalaczony";
      );
      =     L 0.0;
      BLD   103;
      CALL  "Przelaczanie_Stref_K_KB1" (
           Pozycja_Aktualna         := "Pozycja_Aktualna",
           Jazda_Wozka              := L 0.0,
           Strefa_1                 := "Skaner_T_Strefa_1",
           Strefa_2                 := "Skaner_T_Strefa_2",
           Strefa_3                 := "Skaner_T_Strefa_3",
           Strefa_4                 := "Skaner_T_Strefa_4",
           Predkosc_Wozka           := "Predk_Wozka_Kier_KB1");
      NOP   0;
NETWORK
TITLE = Wozek nie jedzie
//Sprawdzenie czy wozek stoi
      A(;
      L     "Predkosc_Aktualna";
      L     0;
      ==I;
      );
      AN    "Zez_Jazda_Wozek";
      =     "Shutte_Stoi";
NETWORK
TITLE =
//Przeniesienie Predkosc aktualnej
      L     "Predkosc_Aktualna";
      T     "Blok_Bledow".Bledy.Predkosc_Aktualna;
      NOP   0;
NETWORK
TITLE =
END_FUNCTION

FUNCTION "Przelaczanie_Stref_K_Rot" : VOID	// FC 102
//Jazda wozka od strony KB1 w kierunku rotacji.Wartosc maja rosnac
//Blok_Stref_Kier_Rot".Wartosc_Pozycji.Poz_0 
//Blok_Stref_Kier_Rot".Wartosc_Pozycji.Poz_1
//Blok_Stref_Kier_Rot".Wartosc_Pozycji.Poz_2
//Blok_Stref_Kier_Rot".Wartosc_Pozycji.Poz_3
//Blok_Stref_Kier_Rot".Wartosc_Pozycji.Poz_4
//Blok_Stref_Kier_Rot".Wartosc_Pozycji.Poz_5
//Blok_Stref_Kier_Rot".Wartosc_Pozycji.Poz_6
//
////*************************************
//
//KB1       
//
//5000               Wozek
//                     |
//                     \/
//
//10000
//
//KB2
//
//
//
//Gender
//15000
//
//
VERSION : 0.1
VAR_INPUT
  Pozycja_Aktualna : DINT ;
  Jazda_Wozka : BOOL ;
END_VAR
VAR_OUTPUT
  Strefa_1 : BOOL ;
  Strefa_2 : BOOL ;
  Strefa_3 : BOOL ;
  Strefa_4 : BOOL ;
  Predkosc_Wozka : INT ;
END_VAR
VAR_TEMP
  Temp_Strefa : DINT ;
  Temp_Predkosc : DINT ;
END_VAR
BEGIN
NETWORK
TITLE =
//Ten Network celowo jest wolny
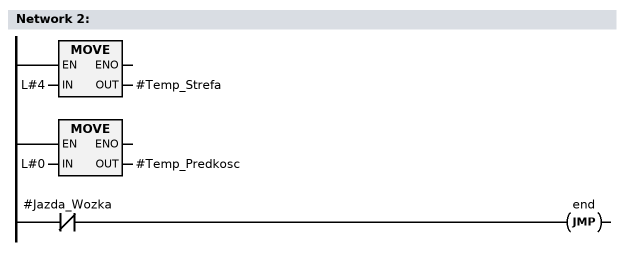
NETWORK
TITLE =
      L     L#4;
      T     #Temp_Strefa;
      L     L#0;
      T     #Temp_Predkosc;
      AN    #Jazda_Wozka;
      JC    end;
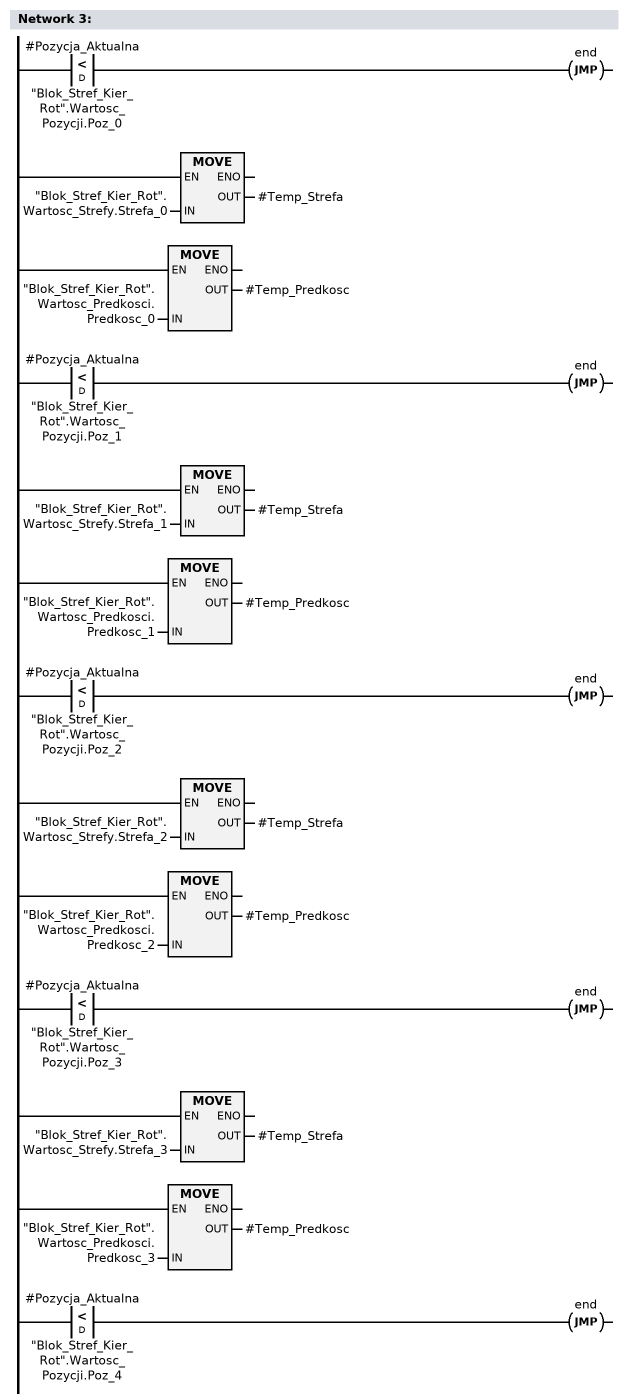
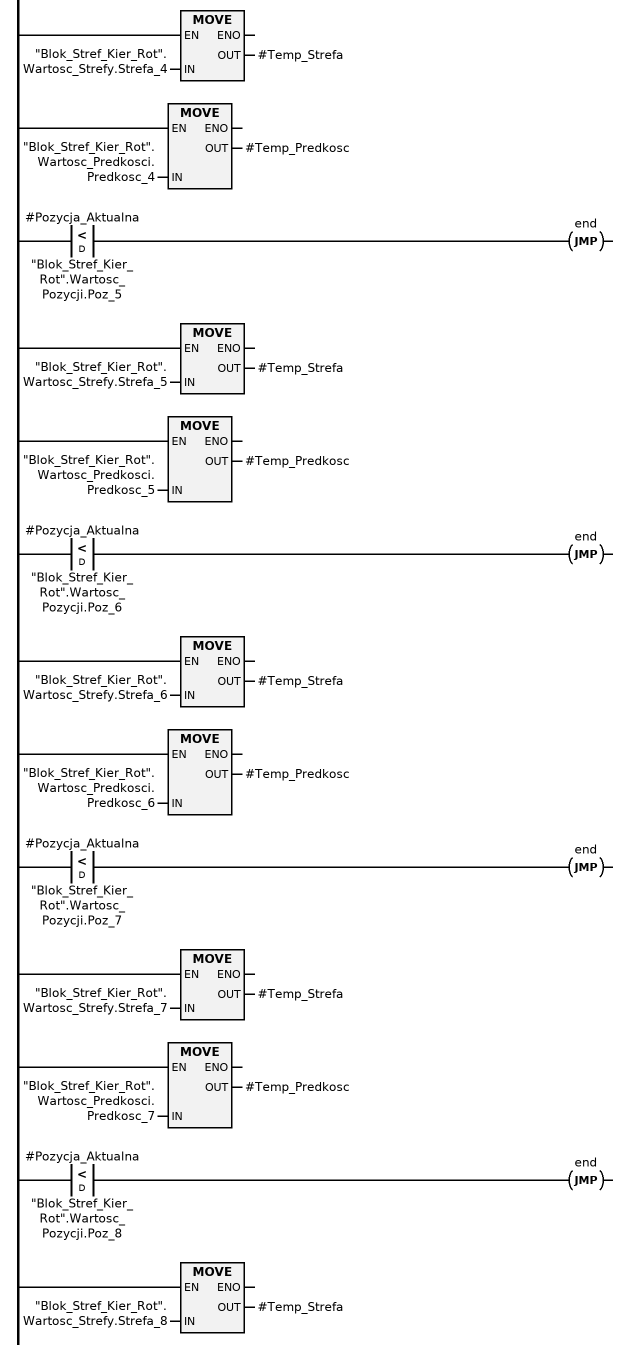
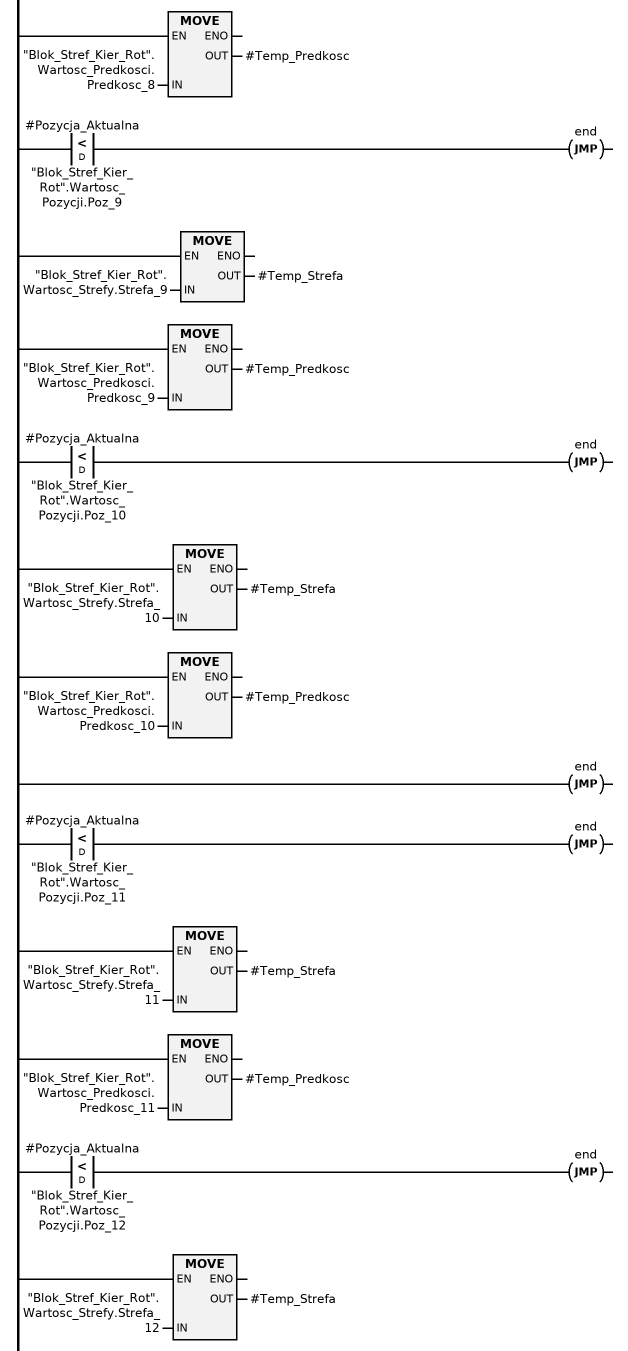
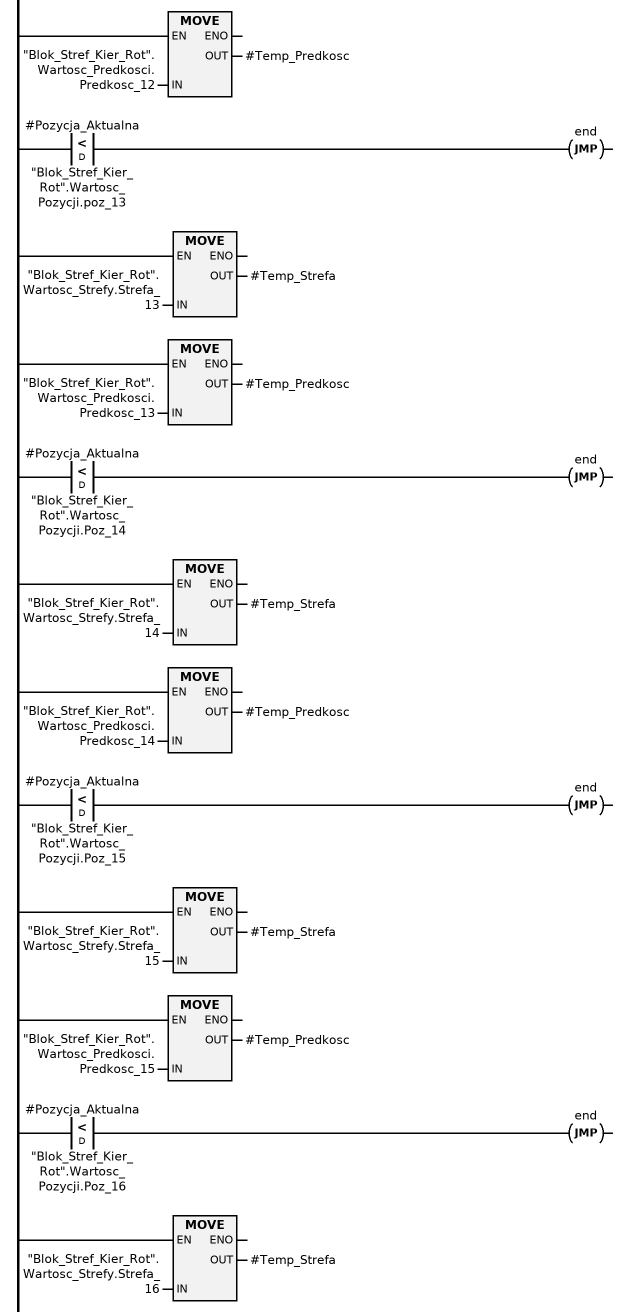
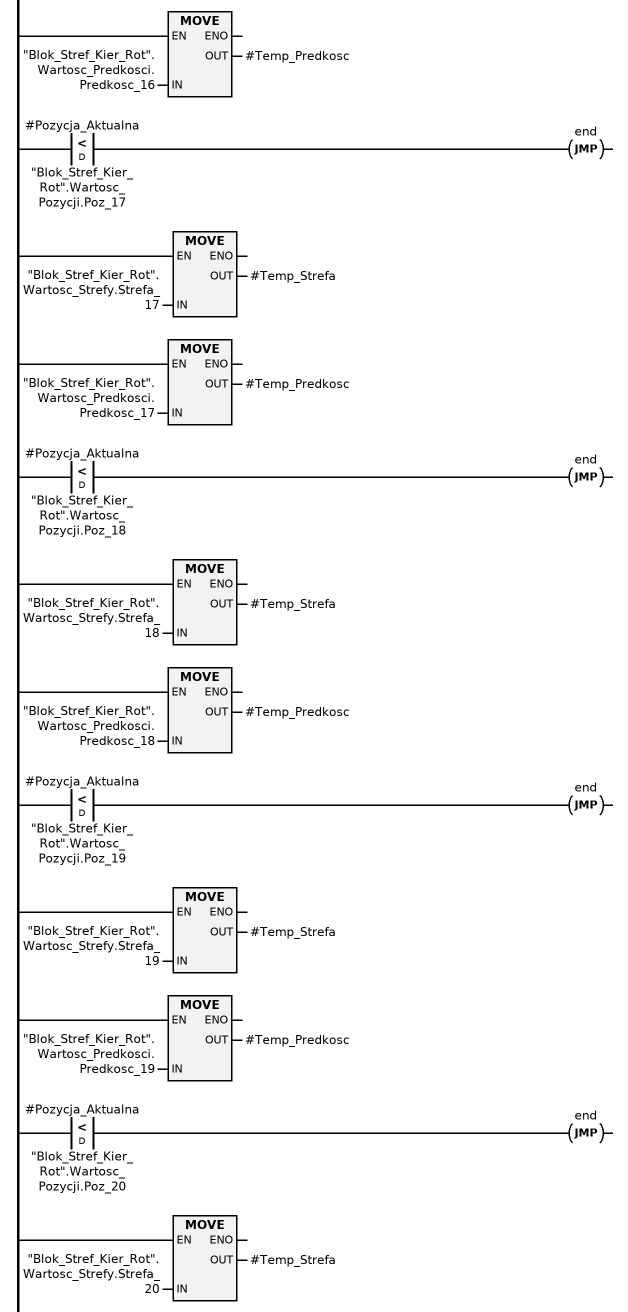
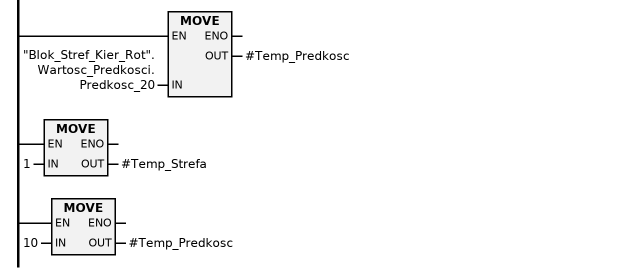
NETWORK
TITLE =
//Porowanie Pozycji z zadana strefa
//KB1       
//
//5000               Wozek
//                     |
//                     \/
//
//10000
//
//KB2
//Strefy :
//skaner przod
//S-Srodek
//G-gora(spedycja)
//
//360-strefa 2 (GS)
//2123-strefa 1(GSD)
//11208-2(GS)
//17550-3(SD)
//*********Poz  0
      L     #Pozycja_Aktualna;	//np 500
      L     "Blok_Stref_Kier_Rot".Wartosc_Pozycji.Poz_0;	//np 320
      <D;
      JC    end;
      L     "Blok_Stref_Kier_Rot".Wartosc_Strefy.Strefa_0;
      T     #Temp_Strefa;
      L     "Blok_Stref_Kier_Rot".Wartosc_Predkosci.Predkosc_0;
      T     #Temp_Predkosc;
//********Poz 1
      L     #Pozycja_Aktualna;	//np 500
      L     "Blok_Stref_Kier_Rot".Wartosc_Pozycji.Poz_1;	// np 400 
      <D;
      JC    end;
      L     "Blok_Stref_Kier_Rot".Wartosc_Strefy.Strefa_1;
      T     #Temp_Strefa;
      L     "Blok_Stref_Kier_Rot".Wartosc_Predkosci.Predkosc_1;
      T     #Temp_Predkosc;
//********Poz 2
      L     #Pozycja_Aktualna;	//500
      L     "Blok_Stref_Kier_Rot".Wartosc_Pozycji.Poz_2;	//600
      <D;
      JC    end;
      L     "Blok_Stref_Kier_Rot".Wartosc_Strefy.Strefa_2;
      T     #Temp_Strefa;
      L     "Blok_Stref_Kier_Rot".Wartosc_Predkosci.Predkosc_2;
      T     #Temp_Predkosc;
//********Poz 3
      L     #Pozycja_Aktualna;	//37000
      L     "Blok_Stref_Kier_Rot".Wartosc_Pozycji.Poz_3;	//40000
      <D;
      JC    end;
      L     "Blok_Stref_Kier_Rot".Wartosc_Strefy.Strefa_3;
      T     #Temp_Strefa;
      L     "Blok_Stref_Kier_Rot".Wartosc_Predkosci.Predkosc_3;
      T     #Temp_Predkosc;
//********Poz 4
      L     #Pozycja_Aktualna;
      L     "Blok_Stref_Kier_Rot".Wartosc_Pozycji.Poz_4;
      <D;
      JC    end;
      L     "Blok_Stref_Kier_Rot".Wartosc_Strefy.Strefa_4;
      T     #Temp_Strefa;
      L     "Blok_Stref_Kier_Rot".Wartosc_Predkosci.Predkosc_4;
      T     #Temp_Predkosc;
//********Poz 5
      L     #Pozycja_Aktualna;
      L     "Blok_Stref_Kier_Rot".Wartosc_Pozycji.Poz_5;
      <D;
      JC    end;
      L     "Blok_Stref_Kier_Rot".Wartosc_Strefy.Strefa_5;
      T     #Temp_Strefa;
      L     "Blok_Stref_Kier_Rot".Wartosc_Predkosci.Predkosc_5;
      T     #Temp_Predkosc;
//********Poz 6
      L     #Pozycja_Aktualna;
      L     "Blok_Stref_Kier_Rot".Wartosc_Pozycji.Poz_6;
      <D;
      JC    end;
      L     "Blok_Stref_Kier_Rot".Wartosc_Strefy.Strefa_6;
      T     #Temp_Strefa;
      L     "Blok_Stref_Kier_Rot".Wartosc_Predkosci.Predkosc_6;
      T     #Temp_Predkosc;
//********Poz 7
      L     #Pozycja_Aktualna;
      L     "Blok_Stref_Kier_Rot".Wartosc_Pozycji.Poz_7;
      <D;
      JC    end;
      L     "Blok_Stref_Kier_Rot".Wartosc_Strefy.Strefa_7;
      T     #Temp_Strefa;
      L     "Blok_Stref_Kier_Rot".Wartosc_Predkosci.Predkosc_7;
      T     #Temp_Predkosc;
//********Poz 8
      L     #Pozycja_Aktualna;
      L     "Blok_Stref_Kier_Rot".Wartosc_Pozycji.Poz_8;
      <D;
      JC    end;
      L     "Blok_Stref_Kier_Rot".Wartosc_Strefy.Strefa_8;
      T     #Temp_Strefa;
      L     "Blok_Stref_Kier_Rot".Wartosc_Predkosci.Predkosc_8;
      T     #Temp_Predkosc;
//********Poz 9
      L     #Pozycja_Aktualna;
      L     "Blok_Stref_Kier_Rot".Wartosc_Pozycji.Poz_9;
      <D;
      JC    end;
      L     "Blok_Stref_Kier_Rot".Wartosc_Strefy.Strefa_9;
      T     #Temp_Strefa;
      L     "Blok_Stref_Kier_Rot".Wartosc_Predkosci.Predkosc_9;
      T     #Temp_Predkosc;
//********Poz 10
      L     #Pozycja_Aktualna;
      L     "Blok_Stref_Kier_Rot".Wartosc_Pozycji.Poz_10;
      <D;
      JC    end;
      L     "Blok_Stref_Kier_Rot".Wartosc_Strefy.Strefa_10;
      T     #Temp_Strefa;
      L     "Blok_Stref_Kier_Rot".Wartosc_Predkosci.Predkosc_10;
      T     #Temp_Predkosc;
      JU    end;
//********Poz 11
      L     #Pozycja_Aktualna;
      L     "Blok_Stref_Kier_Rot".Wartosc_Pozycji.Poz_11;
      <D;
      JC    end;
      L     "Blok_Stref_Kier_Rot".Wartosc_Strefy.Strefa_11;
      T     #Temp_Strefa;
      L     "Blok_Stref_Kier_Rot".Wartosc_Predkosci.Predkosc_11;
      T     #Temp_Predkosc;
//********Poz 12
      L     #Pozycja_Aktualna;
      L     "Blok_Stref_Kier_Rot".Wartosc_Pozycji.Poz_12;
      <D;
      JC    end;
      L     "Blok_Stref_Kier_Rot".Wartosc_Strefy.Strefa_12;
      T     #Temp_Strefa;
      L     "Blok_Stref_Kier_Rot".Wartosc_Predkosci.Predkosc_12;
      T     #Temp_Predkosc;
//********Poz 13
      L     #Pozycja_Aktualna;
      L     "Blok_Stref_Kier_Rot".Wartosc_Pozycji.poz_13;
      <D;
      JC    end;
      L     "Blok_Stref_Kier_Rot".Wartosc_Strefy.Strefa_13;
      T     #Temp_Strefa;
      L     "Blok_Stref_Kier_Rot".Wartosc_Predkosci.Predkosc_13;
      T     #Temp_Predkosc;
//********Poz 14
      L     #Pozycja_Aktualna;
      L     "Blok_Stref_Kier_Rot".Wartosc_Pozycji.Poz_14;
      <D;
      JC    end;
      L     "Blok_Stref_Kier_Rot".Wartosc_Strefy.Strefa_14;
      T     #Temp_Strefa;
      L     "Blok_Stref_Kier_Rot".Wartosc_Predkosci.Predkosc_14;
      T     #Temp_Predkosc;
//********Poz 15
      L     #Pozycja_Aktualna;
      L     "Blok_Stref_Kier_Rot".Wartosc_Pozycji.Poz_15;
      <D;
      JC    end;
      L     "Blok_Stref_Kier_Rot".Wartosc_Strefy.Strefa_15;
      T     #Temp_Strefa;
      L     "Blok_Stref_Kier_Rot".Wartosc_Predkosci.Predkosc_15;
      T     #Temp_Predkosc;
//********Poz 16
      L     #Pozycja_Aktualna;
      L     "Blok_Stref_Kier_Rot".Wartosc_Pozycji.Poz_16;
      <D;
      JC    end;
      L     "Blok_Stref_Kier_Rot".Wartosc_Strefy.Strefa_16;
      T     #Temp_Strefa;
      L     "Blok_Stref_Kier_Rot".Wartosc_Predkosci.Predkosc_16;
      T     #Temp_Predkosc;
//********Poz 17
      L     #Pozycja_Aktualna;
      L     "Blok_Stref_Kier_Rot".Wartosc_Pozycji.Poz_17;
      <D;
      JC    end;
      L     "Blok_Stref_Kier_Rot".Wartosc_Strefy.Strefa_17;
      T     #Temp_Strefa;
      L     "Blok_Stref_Kier_Rot".Wartosc_Predkosci.Predkosc_17;
      T     #Temp_Predkosc;
//********Poz 18
      L     #Pozycja_Aktualna;
      L     "Blok_Stref_Kier_Rot".Wartosc_Pozycji.Poz_18;
      <D;
      JC    end;
      L     "Blok_Stref_Kier_Rot".Wartosc_Strefy.Strefa_18;
      T     #Temp_Strefa;
      L     "Blok_Stref_Kier_Rot".Wartosc_Predkosci.Predkosc_18;
      T     #Temp_Predkosc;
//********Poz 19
      L     #Pozycja_Aktualna;
      L     "Blok_Stref_Kier_Rot".Wartosc_Pozycji.Poz_19;
      <D;
      JC    end;
      L     "Blok_Stref_Kier_Rot".Wartosc_Strefy.Strefa_19;
      T     #Temp_Strefa;
      L     "Blok_Stref_Kier_Rot".Wartosc_Predkosci.Predkosc_19;
      T     #Temp_Predkosc;
//********Poz 20
      L     #Pozycja_Aktualna;
      L     "Blok_Stref_Kier_Rot".Wartosc_Pozycji.Poz_20;
      <D;
      JC    end;
      L     "Blok_Stref_Kier_Rot".Wartosc_Strefy.Strefa_20;
      T     #Temp_Strefa;
      L     "Blok_Stref_Kier_Rot".Wartosc_Predkosci.Predkosc_20;
      T     #Temp_Predkosc;
//Jezeli nic nie wyszlo wybierz strefe najwieksza
      L     1;
      T     #Temp_Strefa;
      L     10;
      T     #Temp_Predkosc;
end:  NOP   0;
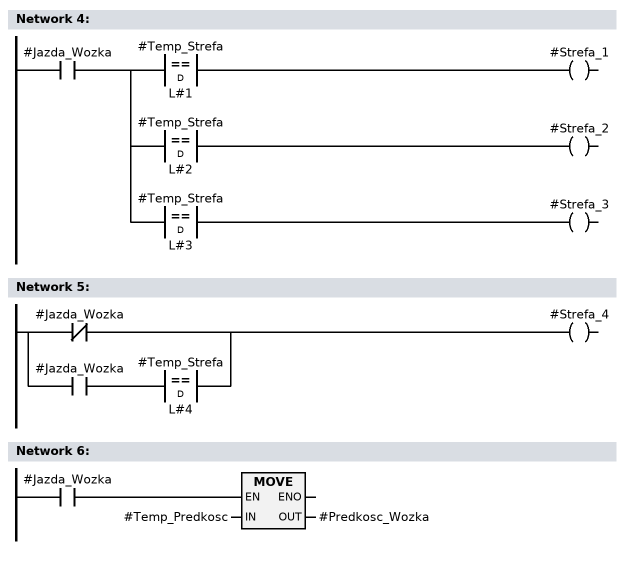
NETWORK
TITLE =
//Przypisanie predkosc. Strefa 1 to strefa podluzna.
//
      A     #Jazda_Wozka;
      =     L 8.0;
      A     L 8.0;
      A(;
      L     #Temp_Strefa;
      L     L#1;
      ==D;
      );
      =     #Strefa_1;
      A     L 8.0;
      A(;
      L     #Temp_Strefa;
      L     L#2;
      ==D;
      );
      =     #Strefa_2;
      A     L 8.0;
      A(;
      L     #Temp_Strefa;
      L     L#3;
      ==D;
      );
      =     #Strefa_3;
NETWORK
TITLE =
//Jezeli wozek stoi
      ON    #Jazda_Wozka;
      O;
      A     #Jazda_Wozka;
      A(;
      L     #Temp_Strefa;
      L     L#4;
      ==D;
      );
      =     #Strefa_4;
NETWORK
TITLE =
//Przyporzadkowanie predkosci
      A     #Jazda_Wozka;
      JNB   _001;
      L     #Temp_Predkosc;
      T     #Predkosc_Wozka;
_001: NOP   0;
END_FUNCTION

FUNCTION "Przelaczanie_Stref_K_KB1" : VOID	// FC 103
//Jazda wozka od strony Rotacji w kierunku KB1. Wartosci wozka maleja
//
VERSION : 0.1
VAR_INPUT
  Pozycja_Aktualna : DINT ;
  Jazda_Wozka : BOOL ;
END_VAR
VAR_OUTPUT
  Strefa_1 : BOOL ;
  Strefa_2 : BOOL ;
  Strefa_3 : BOOL ;
  Strefa_4 : BOOL ;
  Predkosc_Wozka : INT ;
END_VAR
VAR_TEMP
  Temp_Strefa : DINT ;
  Temp_Predkosc : DINT ;
END_VAR
BEGIN
NETWORK
TITLE =
//Ten Network celowo jest wolny
//
//B1       
//
//5000               
//
//10000
//
//KB2
//                        /\
//                        |
//12000                 Wozek
//
//
//Gender
//15000
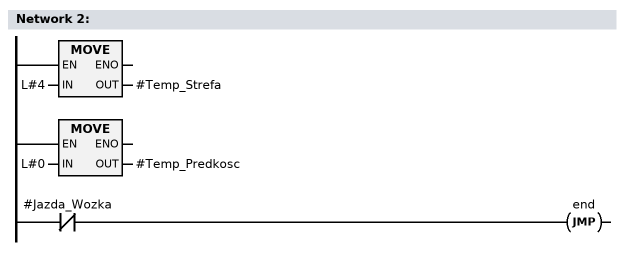
NETWORK
TITLE =
      L     L#4;
      T     #Temp_Strefa;
      L     L#0;
      T     #Temp_Predkosc;
      AN    #Jazda_Wozka;
      JC    end;
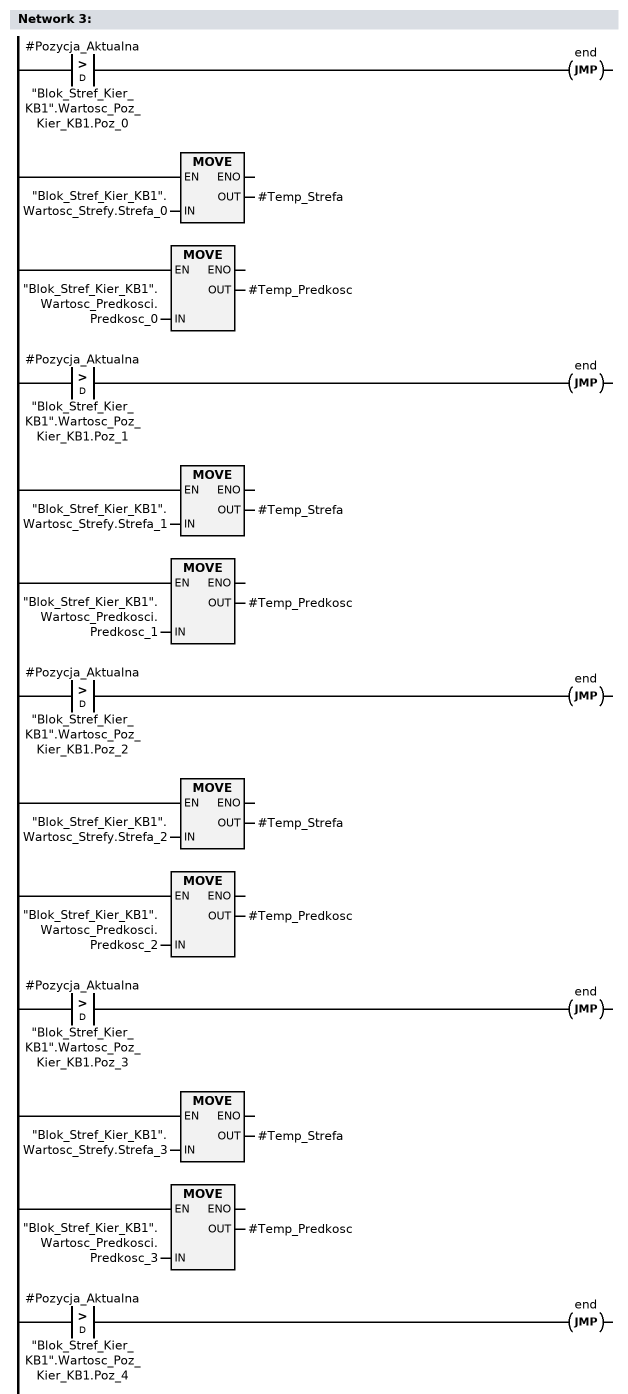
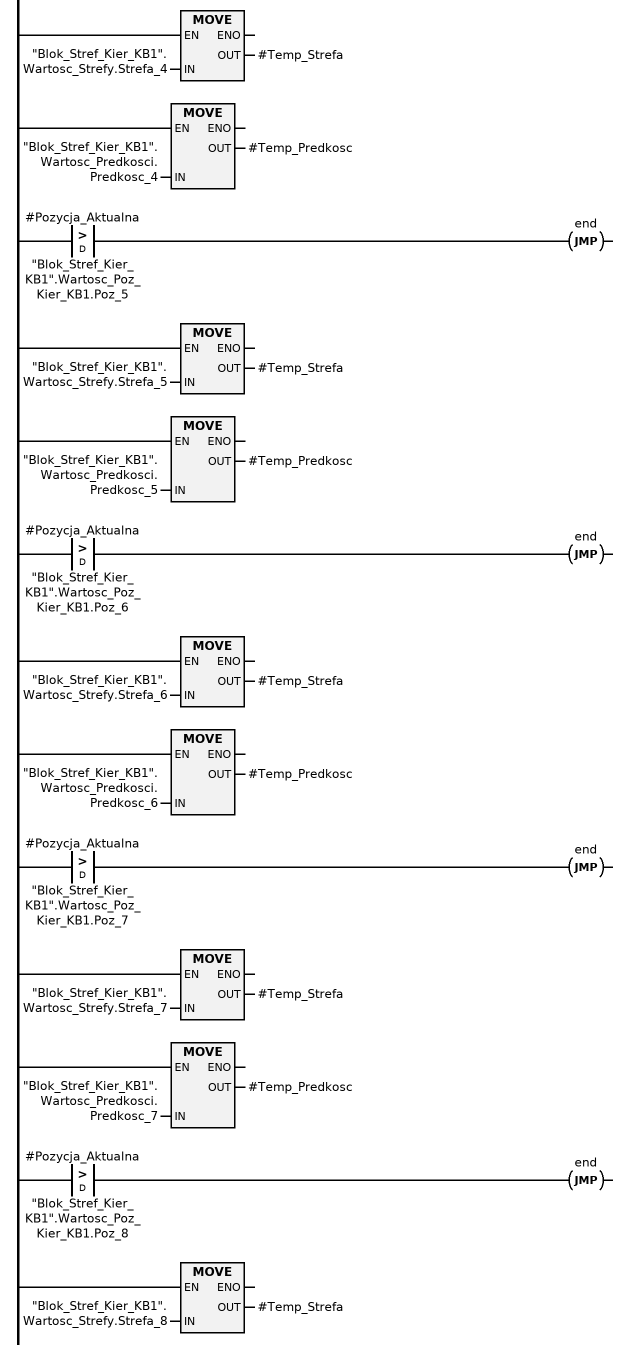
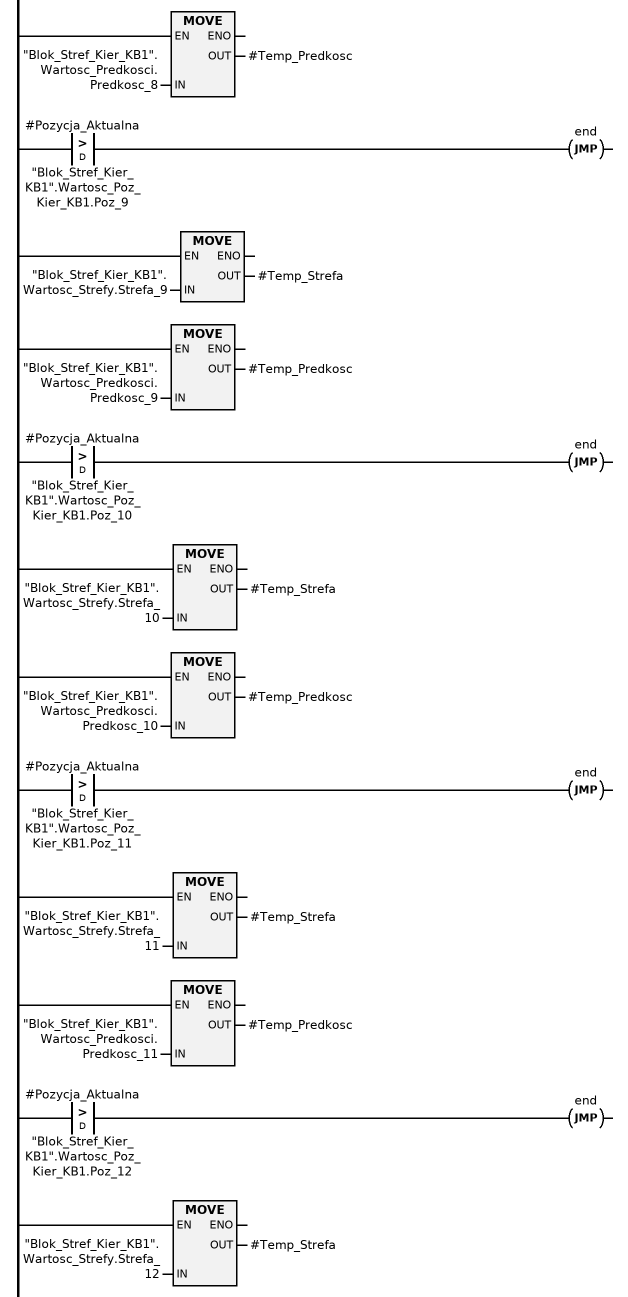
